LIN {X 0,Y 573.248,Z 41.082,A -85,B 0,C 180,E1 -2299.475,E2 -2299.475} C_VEL
LIN {X 0,Y 573.238,Z 41.075,A -85,B 0,C 180,E1 -2302.192,E2 -2302.192} C_VEL
LIN {X 0,Y 573.24,Z 41.084,A -85,B 0,C 180,E1 -2305.229,E2 -2305.229} C_VEL
LIN {X 0,Y 573.243,Z 41.074,A -85,B 0,C 180,E1 -2308.185,E2 -2308.185} C_VEL
LIN {X 0,Y 573.268,Z 41.074,A -85,B 0,C 180,E1 -2310.634,E2 -2310.634} C_VEL
LIN {X 0,Y 573.255,Z 41.08,A -85,B 0,C 180,E1 -2313.024,E2 -2313.024} C_VEL
LIN {X 0,Y 573.279,Z 41.072,A -85,B 0,C 180,E1 -2315.366,E2 -2315.366} C_VEL
LIN {X 0,Y 573.234,Z 41.08,A -85,B 0,C 180,E1 -2318.419,E2 -2318.419} C_VEL
LIN {X 0,Y 573.274,Z 41.078,A -85,B 0,C 180,E1 -2320.731,E2 -2320.731} C_VEL
LIN {X 0,Y 573.252,Z 41.072,A -85,B 0,C 180,E1 -2323.622,E2 -2323.622} C_VEL
LIN {X 0,Y 573.277,Z 41.072,A -85,B 0,C 180,E1 -2325.807,E2 -2325.807} C_VEL
LIN {X 0,Y 573.269,Z 41.074,A -85,B 0,C 180,E1 -2328.745,E2 -2328.745} C_VEL
LIN {X 0,Y 573.288,Z 41.07,A -85,B 0,C 180,E1 -2331.54,E2 -2331.54} C_VEL
LIN {X 0,Y 573.29,Z 41.073,A -85,B 0,C 180,E1 -2334.372,E2 -2334.372} C_VEL
LIN {X 0,Y 573.311,Z 41.074,A -85,B 0,C 180,E1 -2337.892,E2 -2337.892} C_VEL
LIN {X 0,Y 573.332,Z 41.063,A -85,B 0,C 180,E1 -2340.702,E2 -2340.702} C_VEL
LIN {X 0,Y 573.234,Z 41.082,A -85,B 0,C 180,E1 -2343.514,E2 -2343.514} C_VEL
LIN {X 0,Y 573.286,Z 41.078,A -85,B 0,C 180,E1 -2345.628,E2 -2345.628} C_VEL
LIN {X 0,Y 573.275,Z 41.075,A -85,B 0,C 180,E1 -2347.75,E2 -2347.75} C_VEL
LIN {X 0,Y 573.267,Z 41.071,A -85,B 0,C 180,E1 -2350.597,E2 -2350.597} C_VEL
LIN {X 0,Y 573.266,Z 41.073,A -85,B 0,C 180,E1 -2352.748,E2 -2352.748} C_VEL
LIN {X 0,Y 573.239,Z 41.079,A -85,B 0,C 180,E1 -2354.92,E2 -2354.92} C_VEL
LIN {X 0,Y 573.242,Z 41.074,A -85,B 0,C 180,E1 -2357.849,E2 -2357.849} C_VEL
LIN {X 0,Y 573.244,Z 41.074,A -85,B 0,C 180,E1 -2360.077,E2 -2360.077} C_VEL
LIN {X 0,Y 573.236,Z 41.077,A -85,B 0,C 180,E1 -2362.338,E2 -2362.338} C_VEL
LIN {X 0,Y 573.249,Z 41.076,A -85,B 0,C 180,E1 -2364.376,E2 -2364.376} C_VEL
LIN {X 0,Y 572.619,Z 41.161,A -85,B 0,C 180,E1 -2364.962,E2 -2364.962} C_VEL
LIN {X 0,Y 569.76,Z 41.516,A -85,B 0,C 180,E1 -2365.913,E2 -2365.913} C_VEL
LIN {X 0,Y 567.316,Z 41.821,A -85,B 0,C 180,E1 -2366.679,E2 -2366.679} C_VEL
LIN {X 0,Y 566.259,Z 41.946,A -85,B 0,C 180,E1 -2367.27,E2 -2367.27} C_VEL
LIN {X 0,Y 566.171,Z 41.955,A -85,B 0,C 180,E1 -2367.47,E2 -2367.47} C_VEL
LIN {X 0,Y 566.203,Z 41.952,A -85,B 0,C 180,E1 -2369.769,E2 -2369.769} C_VEL
LIN {X 0,Y 566.206,Z 41.959,A -85,B 0,C 180,E1 -2372.43,E2 -2372.43} C_VEL
LIN {X 0,Y 566.172,Z 41.957,A -85,B 0,C 180,E1 -2374.988,E2 -2374.988} C_VEL
LIN {X 0,Y 566.194,Z 41.952,A -85,B 0,C 180,E1 -2377.461,E2 -2377.461} C_VEL
LIN {X 0,Y 566.209,Z 41.957,A -85,B 0,C 180,E1 -2380.199,E2 -2380.199} C_VEL
LIN {X 0,Y 566.197,Z 41.953,A -85,B 0,C 180,E1 -2383.055,E2 -2383.055} C_VEL
LIN {X 0,Y 566.161,Z 41.965,A -85,B 0,C 180,E1 -2386.053,E2 -2386.053} C_VEL
LIN {X 0,Y 566.172,Z 41.956,A -85,B 0,C 180,E1 -2388.86,E2 -2388.86} C_VEL
LIN {X 0,Y 566.204,Z 41.957,A -85,B 0,C 180,E1 -2391.443,E2 -2391.443} C_VEL
LIN {X 0,Y 566.151,Z 41.96,A -85,B 0,C 180,E1 -2394.307,E2 -2394.307} C_VEL
LIN {X 0,Y 566.2,Z 41.955,A -85,B 0,C 180,E1 -2396.896,E2 -2396.896} C_VEL
LIN {X 0,Y 566.17,Z 41.965,A -85,B 0,C 180,E1 -2399.406,E2 -2399.406} C_VEL
LIN {X 0,Y 566.248,Z 42.03,A -85,B 0,C 180,E1 -2402.287,E2 -2402.287} C_VEL
LIN {X 0,Y 566.323,Z 51.031,A -85,B 0,C 180,E1 -2404.059,E2 -2404.059} C_VEL
LIN {X 0,Y 566.238,Z 61.144,A -85,B 0,C 180,E1 -2406.046,E2 -2406.046} C_VEL
LIN {X 0,Y 567.205,Z 67.037,A -85,B 0,C 180,E1 -2406.16,E2 -2406.16} C_VEL
LIN {X 0,Y 566.926,Z 167.119,A -85,B 0,C 180,E1 -2407.448,E2 -2407.448} C_VEL
LIN {X 0,Y 566.828,Z 180.881,A -85,B 0,C 180,E1 -2407.78,E2 -2407.78} C_VEL
LIN {X 0,Y 566.748,Z 192.877,A -85,B 0,C 180,E1 -2408.21,E2 -2408.21} C_VEL
LIN {X 0,Y 566.57,Z 204.986,A -85,B 0,C 180,E1 -2408.797,E2 -2408.797} C_VEL
LIN {X 0,Y 566.416,Z 215.924,A -85,B 0,C 180,E1 -2409.481,E2 -2409.481} C_VEL
LIN {X 0,Y 566.302,Z 226.819,A -85,B 0,C 180,E1 -2410.328,E2 -2410.328} C_VEL
LIN {X 0,Y 566.23,Z 235.633,A -85,B 0,C 180,E1 -2411.173,E2 -2411.173} C_VEL
LIN {X 0,Y 566.102,Z 243.65,A -85,B 0,C 180,E1 -2412.105,E2 -2412.105} C_VEL
LIN {X 0,Y 566.039,Z 251.146,A -85,B 0,C 180,E1 -2413.176,E2 -2413.176} C_VEL
LIN {X 0,Y 565.951,Z 256.676,A -85,B 0,C 180,E1 -2414.145,E2 -2414.145} C_VEL
LIN {X 0,Y 565.943,Z 261.72,A -85,B 0,C 180,E1 -2415.252,E2 -2415.252} C_VEL
LIN {X 0,Y 565.899,Z 265.562,A -85,B 0,C 180,E1 -2416.351,E2 -2416.351} C_VEL
LIN {X 0,Y 565.86,Z 267.528,A -85,B 0,C 180,E1 -2417.082,E2 -2417.082} C_VEL
LIN {X 0,Y 565.869,Z 269.041,A -85,B 0,C 180,E1 -2417.811,E2 -2417.811} C_VEL
LIN {X 0,Y 565.901,Z 270.434,A -85,B 0,C 180,E1 -2418.846,E2 -2418.846} C_VEL
LIN {X 0,Y 565.882,Z 270.993,A -85,B 0,C 180,E1 -2419.987,E2 -2419.987} C_VEL
LIN {X 0,Y 565.829,Z 270.818,A -85,B 0,C 180,E1 -2420.708,E2 -2420.708} C_VEL
LIN {X 0,Y 565.851,Z 270.228,A -85,B 0,C 180,E1 -2421.429,E2 -2421.429} C_VEL
LIN {X 0,Y 565.877,Z 269.245,A -85,B 0,C 180,E1 -2422.148,E2 -2422.148} C_VEL
LIN {X 0,Y 565.945,Z 266.439,A -85,B 0,C 180,E1 -2423.44,E2 -2423.44} C_VEL
LIN {X 0,Y 565.921,Z 262.45,A -85,B 0,C 180,E1 -2424.656,E2 -2424.656} C_VEL
LIN {X 0,Y 565.964,Z 257.776,A -85,B 0,C 180,E1 -2425.727,E2 -2425.727} C_VEL
LIN {X 0,Y 566.004,Z 250.768,A -85,B 0,C 180,E1 -2426.975,E2 -2426.975} C_VEL
LIN {X 0,Y 566.065,Z 243.204,A -85,B 0,C 180,E1 -2428.043,E2 -2428.043} C_VEL
LIN {X 0,Y 566.211,Z 233.725,A -85,B 0,C 180,E1 -2429.111,E2 -2429.111} C_VEL
LIN {X 0,Y 566.297,Z 223.997,A -85,B 0,C 180,E1 -2430,E2 -2430} C_VEL
LIN {X 0,Y 566.443,Z 213.138,A -85,B 0,C 180,E1 -2430.8,E2 -2430.8} C_VEL
LIN {X 0,Y 566.657,Z 200.84,A -85,B 0,C 180,E1 -2431.51,E2 -2431.51} C_VEL
LIN {X 0,Y 566.769,Z 188.815,A -85,B 0,C 180,E1 -2432.043,E2 -2432.043} C_VEL
LIN {X 0,Y 566.841,Z 176.197,A -85,B 0,C 180,E1 -2432.443,E2 -2432.443} C_VEL
LIN {X 0,Y 566.958,Z 162.831,A -85,B 0,C 180,E1 -2432.709,E2 -2432.709} C_VEL
LIN {X 0,Y 567.076,Z 66.314,A -85,B 0,C 180,E1 -2433.942,E2 -2433.942} C_VEL
LIN {X 0,Y 566.213,Z 61.132,A -85,B 0,C 180,E1 -2434.048,E2 -2434.048} C_VEL
LIN {X 0,Y 566.361,Z 48.01,A -85,B 0,C 180,E1 -2436.625,E2 -2436.625} C_VEL
LIN {X 0,Y 566.229,Z 41.953,A -85,B 0,C 180,E1 -2437.847,E2 -2437.847} C_VEL
LIN {X 0,Y 566.24,Z 41.956,A -85,B 0,C 180,E1 -2440.73,E2 -2440.73} C_VEL
LIN {X 0,Y 566.21,Z 41.955,A -85,B 0,C 180,E1 -2442.91,E2 -2442.91} C_VEL
LIN {X 0,Y 566.201,Z 41.953,A -85,B 0,C 180,E1 -2445.11,E2 -2445.11} C_VEL
LIN {X 0,Y 566.202,Z 41.951,A -85,B 0,C 180,E1 -2447.332,E2 -2447.332} C_VEL
LIN {X 0,Y 566.21,Z 41.96,A -85,B 0,C 180,E1 -2450.338,E2 -2450.338} C_VEL
LIN {X 0,Y 566.171,Z 41.955,A -85,B 0,C 180,E1 -2453.281,E2 -2453.281} C_VEL
LIN {X 0,Y 566.215,Z 41.953,A -85,B 0,C 180,E1 -2455.749,E2 -2455.749} C_VEL
LIN {X 0,Y 566.205,Z 41.958,A -85,B 0,C 180,E1 -2458.202,E2 -2458.202} C_VEL
LIN {X 0,Y 566.193,Z 41.952,A -85,B 0,C 180,E1 -2461.077,E2 -2461.077} C_VEL
LIN {X 0,Y 566.215,Z 41.957,A -85,B 0,C 180,E1 -2463.734,E2 -2463.734} C_VEL
LIN {X 0,Y 566.21,Z 41.951,A -85,B 0,C 180,E1 -2466.57,E2 -2466.57} C_VEL
LIN {X 0,Y 566.219,Z 41.959,A -85,B 0,C 180,E1 -2469.686,E2 -2469.686} C_VEL
LIN {X 0,Y 566.204,Z 41.952,A -85,B 0,C 180,E1 -2472.917,E2 -2472.917} C_VEL
LIN {X 0,Y 566.197,Z 41.953,A -85,B 0,C 180,E1 -2476.05,E2 -2476.05} C_VEL
LIN {X 0,Y 566.207,Z 41.958,A -85,B 0,C 180,E1 -2479.215,E2 -2479.215} C_VEL
LIN {X 0,Y 566.189,Z 41.956,A -85,B 0,C 180,E1 -2481.637,E2 -2481.637} C_VEL
LIN {X 0,Y 566.167,Z 41.956,A -85,B 0,C 180,E1 -2484.308,E2 -2484.308} C_VEL
LIN {X 0,Y 566.224,Z 41.956,A -85,B 0,C 180,E1 -2486.898,E2 -2486.898} C_VEL
LIN {X 0,Y 566.185,Z 41.956,A -85,B 0,C 180,E1 -2489.407,E2 -2489.407} C_VEL
LIN {X 0,Y 566.217,Z 41.949,A -85,B 0,C 180,E1 -2491.858,E2 -2491.858} C_VEL
LIN {X 0,Y 566.214,Z 41.952,A -85,B 0,C 180,E1 -2494.251,E2 -2494.251} C_VEL
LIN {X 0,Y 566.178,Z 41.964,A -85,B 0,C 180,E1 -2496.719,E2 -2496.719} C_VEL
LIN {X 0,Y 566.212,Z 41.95,A -85,B 0,C 180,E1 -2499.663,E2 -2499.663} C_VEL
LIN {X 0,Y 566.203,Z 41.957,A -85,B 0,C 180,E1 -2502.669,E2 -2502.669} C_VEL
LIN {X 0,Y 566.24,Z 41.947,A -85,B 0,C 180,E1 -2505.627,E2 -2505.627} C_VEL
LIN {X 0,Y 566.241,Z 41.95,A -85,B 0,C 180,E1 -2508.675,E2 -2508.675} C_VEL
LIN {X 0,Y 566.212,Z 41.951,A -85,B 0,C 180,E1 -2511.434,E2 -2511.434} C_VEL
LIN {X 0,Y 566.259,Z 41.95,A -85,B 0,C 180,E1 -2514.302,E2 -2514.302} C_VEL
LIN {X 0,Y 566.284,Z 41.95,A -85,B 0,C 180,E1 -2517.866,E2 -2517.866} C_VEL
LIN {X 0,Y 566.304,Z 41.939,A -85,B 0,C 180,E1 -2520.711,E2 -2520.711} C_VEL
LIN {X 0,Y 566.273,Z 41.942,A -85,B 0,C 180,E1 -2522.846,E2 -2522.846} C_VEL
LIN {X 0,Y 566.255,Z 41.953,A -85,B 0,C 180,E1 -2525.698,E2 -2525.698} C_VEL
LIN {X 0,Y 566.211,Z 41.95,A -85,B 0,C 180,E1 -2528.566,E2 -2528.566} C_VEL
LIN {X 0,Y 566.248,Z 41.955,A -85,B 0,C 180,E1 -2531.454,E2 -2531.454} C_VEL
LIN {X 0,Y 566.236,Z 41.947,A -85,B 0,C 180,E1 -2534.504,E2 -2534.504} C_VEL
LIN {X 0,Y 566.204,Z 41.959,A -85,B 0,C 180,E1 -2537.332,E2 -2537.332} C_VEL
LIN {X 0,Y 566.212,Z 41.95,A -85,B 0,C 180,E1 -2540.337,E2 -2540.337} C_VEL
LIN {X 0,Y 566.174,Z 41.96,A -85,B 0,C 180,E1 -2543.281,E2 -2543.281} C_VEL
LIN {X 0,Y 566.211,Z 41.95,A -85,B 0,C 180,E1 -2545.749,E2 -2545.749} C_VEL
LIN {X 0,Y 566.209,Z 41.952,A -85,B 0,C 180,E1 -2548.202,E2 -2548.202} C_VEL
LIN {X 0,Y 566.195,Z 41.956,A -85,B 0,C 180,E1 -2551.076,E2 -2551.076} C_VEL
LIN {X 0,Y 566.201,Z 41.951,A -85,B 0,C 180,E1 -2553.732,E2 -2553.732} C_VEL
LIN {X 0,Y 566.187,Z 41.962,A -85,B 0,C 180,E1 -2556.571,E2 -2556.571} C_VEL
LIN {X 0,Y 566.218,Z 41.95,A -85,B 0,C 180,E1 -2559.685,E2 -2559.685} C_VEL
LIN {X 0,Y 566.205,Z 41.952,A -85,B 0,C 180,E1 -2562.917,E2 -2562.917} C_VEL
LIN {X 0,Y 566.164,Z 41.962,A -85,B 0,C 180,E1 -2565.96,E2 -2565.96} C_VEL
LIN {X 0,Y 566.19,Z 41.962,A -85,B 0,C 180,E1 -2568.139,E2 -2568.139} C_VEL
LIN {X 0,Y 566.214,Z 41.95,A -85,B 0,C 180,E1 -2570.726,E2 -2570.726} C_VEL
LIN {X 0,Y 566.186,Z 41.956,A -85,B 0,C 180,E1 -2573.429,E2 -2573.429} C_VEL
LIN {X 0,Y 566.201,Z 41.954,A -85,B 0,C 180,E1 -2576.268,E2 -2576.268} C_VEL
LIN {X 0,Y 566.191,Z 41.953,A -85,B 0,C 180,E1 -2578.924,E2 -2578.924} C_VEL
LIN {X 0,Y 566.216,Z 41.956,A -85,B 0,C 180,E1 -2581.857,E2 -2581.857} C_VEL
LIN {X 0,Y 566.21,Z 41.953,A -85,B 0,C 180,E1 -2584.251,E2 -2584.251} C_VEL
LIN {X 0,Y 566.261,Z 42.121,A -85,B 0,C 180,E1 -2585.676,E2 -2585.676} C_VEL
LIN {X 0,Y 567.074,Z 47.877,A -85,B 0,C 180,E1 -2586.508,E2 -2586.508} C_VEL
LIN {X 0,Y 566.844,Z 66.903,A -85,B 0,C 180,E1 -2589.117,E2 -2589.117} C_VEL
LIN {X 0,Y 566.689,Z 87.816,A -85,B 0,C 180,E1 -2591.938,E2 -2591.938} C_VEL
LIN {X 0,Y 566.434,Z 110.041,A -85,B 0,C 180,E1 -2594.897,E2 -2594.897} C_VEL
LIN {X 0,Y 566.431,Z 118.274,A -85,B 0,C 180,E1 -2595.987,E2 -2595.987} C_VEL
LIN {X 0,Y 567.176,Z 125.162,A -85,B 0,C 180,E1 -2596.095,E2 -2596.095} C_VEL
LIN {X 0,Y 566.941,Z 226.937,A -85,B 0,C 180,E1 -2597.402,E2 -2597.402} C_VEL
LIN {X 0,Y 566.859,Z 240.211,A -85,B 0,C 180,E1 -2597.719,E2 -2597.719} C_VEL
LIN {X 0,Y 566.761,Z 252.373,A -85,B 0,C 180,E1 -2598.148,E2 -2598.148} C_VEL
LIN {X 0,Y 566.604,Z 264.236,A -85,B 0,C 180,E1 -2598.712,E2 -2598.712} C_VEL
LIN {X 0,Y 566.442,Z 276.192,A -85,B 0,C 180,E1 -2599.455,E2 -2599.455} C_VEL
LIN {X 0,Y 566.325,Z 286.604,A -85,B 0,C 180,E1 -2600.265,E2 -2600.265} C_VEL
LIN {X 0,Y 566.207,Z 295.112,A -85,B 0,C 180,E1 -2601.074,E2 -2601.074} C_VEL
LIN {X 0,Y 566.112,Z 302.96,A -85,B 0,C 180,E1 -2601.972,E2 -2601.972} C_VEL
LIN {X 0,Y 566.004,Z 310.622,A -85,B 0,C 180,E1 -2603.047,E2 -2603.047} C_VEL
LIN {X 0,Y 566.004,Z 317.679,A -85,B 0,C 180,E1 -2604.299,E2 -2604.299} C_VEL
LIN {X 0,Y 565.933,Z 322.372,A -85,B 0,C 180,E1 -2605.37,E2 -2605.37} C_VEL
LIN {X 0,Y 565.927,Z 325.958,A -85,B 0,C 180,E1 -2606.44,E2 -2606.44} C_VEL
LIN {X 0,Y 565.878,Z 327.807,A -85,B 0,C 180,E1 -2607.152,E2 -2607.152} C_VEL
LIN {X 0,Y 565.846,Z 330.183,A -85,B 0,C 180,E1 -2608.577,E2 -2608.577} C_VEL
LIN {X 0,Y 565.839,Z 331,A -85,B 0,C 180,E1 -2610,E2 -2610} C_VEL
LIN {X 0,Y 565.846,Z 330.185,A -85,B 0,C 180,E1 -2611.423,E2 -2611.423} C_VEL
LIN {X 0,Y 565.878,Z 327.81,A -85,B 0,C 180,E1 -2612.848,E2 -2612.848} C_VEL
LIN {X 0,Y 565.926,Z 324.895,A -85,B 0,C 180,E1 -2613.916,E2 -2613.916} C_VEL
LIN {X 0,Y 565.878,Z 320.948,A -85,B 0,C 180,E1 -2614.987,E2 -2614.987} C_VEL
LIN {X 0,Y 566.004,Z 315.867,A -85,B 0,C 180,E1 -2616.058,E2 -2616.058} C_VEL
LIN {X 0,Y 566.04,Z 309.467,A -85,B 0,C 180,E1 -2617.132,E2 -2617.132} C_VEL
LIN {X 0,Y 566.134,Z 301.477,A -85,B 0,C 180,E1 -2618.208,E2 -2618.208} C_VEL
LIN {X 0,Y 566.229,Z 293.333,A -85,B 0,C 180,E1 -2619.105,E2 -2619.105} C_VEL
LIN {X 0,Y 566.342,Z 283.397,A -85,B 0,C 180,E1 -2620.005,E2 -2620.005} C_VEL
LIN {X 0,Y 566.512,Z 272.289,A -85,B 0,C 180,E1 -2620.808,E2 -2620.808} C_VEL
LIN {X 0,Y 566.613,Z 261.17,A -85,B 0,C 180,E1 -2621.447,E2 -2621.447} C_VEL
LIN {X 0,Y 566.748,Z 248.975,A -85,B 0,C 180,E1 -2621.988,E2 -2621.988} C_VEL
LIN {X 0,Y 566.887,Z 236.171,A -85,B 0,C 180,E1 -2622.394,E2 -2622.394} C_VEL
LIN {X 0,Y 566.991,Z 224.1,A -85,B 0,C 180,E1 -2622.642,E2 -2622.642} C_VEL
LIN {X 0,Y 567.07,Z 122.848,A -85,B 0,C 180,E1 -2623.937,E2 -2623.937} C_VEL
LIN {X 0,Y 566.43,Z 118.181,A -85,B 0,C 180,E1 -2624.024,E2 -2624.024} C_VEL
LIN {X 0,Y 566.583,Z 96.455,A -85,B 0,C 180,E1 -2626.903,E2 -2626.903} C_VEL
LIN {X 0,Y 566.791,Z 75.206,A -85,B 0,C 180,E1 -2629.748,E2 -2629.748} C_VEL
LIN {X 0,Y 566.965,Z 54.285,A -85,B 0,C 180,E1 -2632.599,E2 -2632.599} C_VEL
LIN {X 0,Y 566.958,Z 45.846,A -85,B 0,C 180,E1 -2633.766,E2 -2633.766} C_VEL
LIN {X 0,Y 566.257,Z 41.954,A -85,B 0,C 180,E1 -2634.349,E2 -2634.349} C_VEL
LIN {X 0,Y 566.211,Z 41.952,A -85,B 0,C 180,E1 -2637.339,E2 -2637.339} C_VEL
LIN {X 0,Y 566.204,Z 41.954,A -85,B 0,C 180,E1 -2639.769,E2 -2639.769} C_VEL
LIN {X 0,Y 566.206,Z 41.957,A -85,B 0,C 180,E1 -2642.43,E2 -2642.43} C_VEL
LIN {X 0,Y 566.184,Z 41.954,A -85,B 0,C 180,E1 -2644.99,E2 -2644.99} C_VEL
LIN {X 0,Y 566.199,Z 41.954,A -85,B 0,C 180,E1 -2647.461,E2 -2647.461} C_VEL
LIN {X 0,Y 566.21,Z 41.955,A -85,B 0,C 180,E1 -2650.199,E2 -2650.199} C_VEL
LIN {X 0,Y 566.203,Z 41.952,A -85,B 0,C 180,E1 -2653.054,E2 -2653.054} C_VEL
LIN {X 0,Y 566.197,Z 41.955,A -85,B 0,C 180,E1 -2656.049,E2 -2656.049} C_VEL
LIN {X 0,Y 566.207,Z 41.955,A -85,B 0,C 180,E1 -2659.215,E2 -2659.215} C_VEL
LIN {X 0,Y 566.189,Z 41.958,A -85,B 0,C 180,E1 -2661.637,E2 -2661.637} C_VEL
LIN {X 0,Y 566.167,Z 41.955,A -85,B 0,C 180,E1 -2664.308,E2 -2664.308} C_VEL
LIN {X 0,Y 566.207,Z 41.955,A -85,B 0,C 180,E1 -2666.897,E2 -2666.897} C_VEL
LIN {X 0,Y 566.185,Z 41.957,A -85,B 0,C 180,E1 -2669.407,E2 -2669.407} C_VEL
LIN {X 0,Y 566.217,Z 41.95,A -85,B 0,C 180,E1 -2671.857,E2 -2671.857} C_VEL
LIN {X 0,Y 566.214,Z 41.95,A -85,B 0,C 180,E1 -2674.251,E2 -2674.251} C_VEL
LIN {X 0,Y 566.174,Z 41.964,A -85,B 0,C 180,E1 -2676.719,E2 -2676.719} C_VEL
LIN {X 0,Y 566.212,Z 41.95,A -85,B 0,C 180,E1 -2679.663,E2 -2679.663} C_VEL
LIN {X 0,Y 566.203,Z 41.957,A -85,B 0,C 180,E1 -2682.668,E2 -2682.668} C_VEL
LIN {X 0,Y 566.239,Z 41.947,A -85,B 0,C 180,E1 -2685.627,E2 -2685.627} C_VEL
LIN {X 0,Y 566.241,Z 41.95,A -85,B 0,C 180,E1 -2688.675,E2 -2688.675} C_VEL
LIN {X 0,Y 566.232,Z 41.948,A -85,B 0,C 180,E1 -2691.434,E2 -2691.434} C_VEL
LIN {X 0,Y 566.259,Z 41.95,A -85,B 0,C 180,E1 -2694.302,E2 -2694.302} C_VEL
LIN {X 0,Y 566.283,Z 41.949,A -85,B 0,C 180,E1 -2697.866,E2 -2697.866} C_VEL
LIN {X 0,Y 566.303,Z 41.939,A -85,B 0,C 180,E1 -2700.711,E2 -2700.711} C_VEL
LIN {X 0,Y 566.272,Z 41.942,A -85,B 0,C 180,E1 -2702.845,E2 -2702.845} C_VEL
LIN {X 0,Y 566.253,Z 41.953,A -85,B 0,C 180,E1 -2705.698,E2 -2705.698} C_VEL
LIN {X 0,Y 566.209,Z 41.949,A -85,B 0,C 180,E1 -2708.566,E2 -2708.566} C_VEL
LIN {X 0,Y 566.247,Z 41.954,A -85,B 0,C 180,E1 -2711.454,E2 -2711.454} C_VEL
LIN {X 0,Y 566.234,Z 41.947,A -85,B 0,C 180,E1 -2714.504,E2 -2714.504} C_VEL
LIN {X 0,Y 566.202,Z 41.957,A -85,B 0,C 180,E1 -2717.332,E2 -2717.332} C_VEL
LIN {X 0,Y 566.211,Z 41.951,A -85,B 0,C 180,E1 -2720.337,E2 -2720.337} C_VEL
LIN {X 0,Y 566.172,Z 41.958,A -85,B 0,C 180,E1 -2723.28,E2 -2723.28} C_VEL
LIN {X 0,Y 566.208,Z 41.951,A -85,B 0,C 180,E1 -2725.749,E2 -2725.749} C_VEL
LIN {X 0,Y 566.171,Z 41.955,A -85,B 0,C 180,E1 -2727.47,E2 -2727.47} C_VEL
LIN {X 0,Y 565.5,Z 42.041,A -85,B 0,C 180,E1 -2728.064,E2 -2728.064} C_VEL
LIN {X 0,Y 562.649,Z 42.398,A -85,B 0,C 180,E1 -2729.028,E2 -2729.028} C_VEL
LIN {X 0,Y 560.247,Z 42.696,A -85,B 0,C 180,E1 -2729.804,E2 -2729.804} C_VEL
LIN {X 0,Y 559.221,Z 42.828,A -85,B 0,C 180,E1 -2730.403,E2 -2730.403} C_VEL
LIN {X 0,Y 559.141,Z 42.832,A -85,B 0,C 180,E1 -2730.606,E2 -2730.606} C_VEL
LIN {X 0,Y 559.156,Z 42.835,A -85,B 0,C 180,E1 -2732.715,E2 -2732.715} C_VEL
LIN {X 0,Y 559.121,Z 42.834,A -85,B 0,C 180,E1 -2735.325,E2 -2735.325} C_VEL
LIN {X 0,Y 559.132,Z 42.837,A -85,B 0,C 180,E1 -2738.018,E2 -2738.018} C_VEL
LIN {X 0,Y 559.156,Z 42.828,A -85,B 0,C 180,E1 -2740.812,E2 -2740.812} C_VEL
LIN {X 0,Y 559.138,Z 42.837,A -85,B 0,C 180,E1 -2743.734,E2 -2743.734} C_VEL
LIN {X 0,Y 559.133,Z 42.833,A -85,B 0,C 180,E1 -2746.805,E2 -2746.805} C_VEL
LIN {X 0,Y 559.157,Z 42.831,A -85,B 0,C 180,E1 -2749.187,E2 -2749.187} C_VEL
LIN {X 0,Y 559.127,Z 42.839,A -85,B 0,C 180,E1 -2751.982,E2 -2751.982} C_VEL
LIN {X 0,Y 559.13,Z 42.834,A -85,B 0,C 180,E1 -2754.788,E2 -2754.788} C_VEL
LIN {X 0,Y 559.154,Z 42.839,A -85,B 0,C 180,E1 -2757.365,E2 -2757.365} C_VEL
LIN {X 0,Y 559.12,Z 42.837,A -85,B 0,C 180,E1 -2760.148,E2 -2760.148} C_VEL
LIN {X 0,Y 559.225,Z 42.921,A -85,B 0,C 180,E1 -2762.19,E2 -2762.19} C_VEL
LIN {X 0,Y 559.332,Z 49.619,A -85,B 0,C 180,E1 -2763.524,E2 -2763.524} C_VEL
LIN {X 0,Y 559.216,Z 61.527,A -85,B 0,C 180,E1 -2765.878,E2 -2765.878} C_VEL
LIN {X 0,Y 560.309,Z 68.487,A -85,B 0,C 180,E1 -2766,E2 -2766} C_VEL
LIN {X 0,Y 559.997,Z 167.977,A -85,B 0,C 180,E1 -2767.299,E2 -2767.299} C_VEL
LIN {X 0,Y 559.923,Z 181.603,A -85,B 0,C 180,E1 -2767.637,E2 -2767.637} C_VEL
LIN {X 0,Y 559.809,Z 193.573,A -85,B 0,C 180,E1 -2768.075,E2 -2768.075} C_VEL
LIN {X 0,Y 559.626,Z 205.125,A -85,B 0,C 180,E1 -2768.642,E2 -2768.642} C_VEL
LIN {X 0,Y 559.456,Z 215.753,A -85,B 0,C 180,E1 -2769.31,E2 -2769.31} C_VEL
LIN {X 0,Y 559.327,Z 226.671,A -85,B 0,C 180,E1 -2770.168,E2 -2770.168} C_VEL
LIN {X 0,Y 559.208,Z 236.374,A -85,B 0,C 180,E1 -2771.118,E2 -2771.118} C_VEL
LIN {X 0,Y 559.039,Z 244.23,A -85,B 0,C 180,E1 -2772.061,E2 -2772.061} C_VEL
LIN {X 0,Y 558.957,Z 251.861,A -85,B 0,C 180,E1 -2773.191,E2 -2773.191} C_VEL
LIN {X 0,Y 558.865,Z 257.92,A -85,B 0,C 180,E1 -2774.313,E2 -2774.313} C_VEL
LIN {X 0,Y 558.826,Z 263.113,A -85,B 0,C 180,E1 -2775.554,E2 -2775.554} C_VEL
LIN {X 0,Y 558.763,Z 267.208,A -85,B 0,C 180,E1 -2776.915,E2 -2776.915} C_VEL
LIN {X 0,Y 558.777,Z 268.806,A -85,B 0,C 180,E1 -2777.654,E2 -2777.654} C_VEL
LIN {X 0,Y 558.798,Z 270.417,A -85,B 0,C 180,E1 -2778.815,E2 -2778.815} C_VEL
LIN {X 0,Y 558.778,Z 270.965,A -85,B 0,C 180,E1 -2779.858,E2 -2779.858} C_VEL
LIN {X 0,Y 558.74,Z 270.885,A -85,B 0,C 180,E1 -2780.589,E2 -2780.589} C_VEL
LIN {X 0,Y 558.765,Z 270.368,A -85,B 0,C 180,E1 -2781.319,E2 -2781.319} C_VEL
LIN {X 0,Y 558.795,Z 269.441,A -85,B 0,C 180,E1 -2782.048,E2 -2782.048} C_VEL
LIN {X 0,Y 558.844,Z 266.487,A -85,B 0,C 180,E1 -2783.464,E2 -2783.464} C_VEL
LIN {X 0,Y 558.845,Z 262.934,A -85,B 0,C 180,E1 -2784.588,E2 -2784.588} C_VEL
LIN {X 0,Y 558.892,Z 258.419,A -85,B 0,C 180,E1 -2785.673,E2 -2785.673} C_VEL
LIN {X 0,Y 558.911,Z 251.637,A -85,B 0,C 180,E1 -2786.937,E2 -2786.937} C_VEL
LIN {X 0,Y 559,Z 244.308,A -85,B 0,C 180,E1 -2788.019,E2 -2788.019} C_VEL
LIN {X 0,Y 559.167,Z 236.838,A -85,B 0,C 180,E1 -2788.92,E2 -2788.92} C_VEL
LIN {X 0,Y 559.265,Z 227.84,A -85,B 0,C 180,E1 -2789.82,E2 -2789.82} C_VEL
LIN {X 0,Y 559.394,Z 217.864,A -85,B 0,C 180,E1 -2790.63,E2 -2790.63} C_VEL
LIN {X 0,Y 559.62,Z 206.803,A -85,B 0,C 180,E1 -2791.349,E2 -2791.349} C_VEL
LIN {X 0,Y 559.803,Z 194.425,A -85,B 0,C 180,E1 -2791.979,E2 -2791.979} C_VEL
LIN {X 0,Y 559.895,Z 181.704,A -85,B 0,C 180,E1 -2792.451,E2 -2792.451} C_VEL
LIN {X 0,Y 560.034,Z 168.079,A -85,B 0,C 180,E1 -2792.787,E2 -2792.787} C_VEL
LIN {X 0,Y 560.184,Z 66.835,A -85,B 0,C 180,E1 -2794.114,E2 -2794.114} C_VEL
LIN {X 0,Y 559.194,Z 61.429,A -85,B 0,C 180,E1 -2794.235,E2 -2794.235} C_VEL
LIN {X 0,Y 559.377,Z 48.905,A -85,B 0,C 180,E1 -2796.705,E2 -2796.705} C_VEL
LIN {X 0,Y 559.206,Z 42.829,A -85,B 0,C 180,E1 -2797.924,E2 -2797.924} C_VEL
LIN {X 0,Y 559.197,Z 42.831,A -85,B 0,C 180,E1 -2800.867,E2 -2800.867} C_VEL
LIN {X 0,Y 559.173,Z 42.827,A -85,B 0,C 180,E1 -2803.816,E2 -2803.816} C_VEL
LIN {X 0,Y 559.183,Z 42.83,A -85,B 0,C 180,E1 -2806.803,E2 -2806.803} C_VEL
LIN {X 0,Y 559.168,Z 42.829,A -85,B 0,C 180,E1 -2809.838,E2 -2809.838} C_VEL
LIN {X 0,Y 559.144,Z 42.838,A -85,B 0,C 180,E1 -2812.153,E2 -2812.153} C_VEL
LIN {X 0,Y 559.178,Z 42.826,A -85,B 0,C 180,E1 -2815.298,E2 -2815.298} C_VEL
LIN {X 0,Y 559.184,Z 42.829,A -85,B 0,C 180,E1 -2817.712,E2 -2817.712} C_VEL
LIN {X 0,Y 559.156,Z 42.836,A -85,B 0,C 180,E1 -2820.183,E2 -2820.183} C_VEL
LIN {X 0,Y 559.159,Z 42.829,A -85,B 0,C 180,E1 -2822.715,E2 -2822.715} C_VEL
LIN {X 0,Y 559.147,Z 42.832,A -85,B 0,C 180,E1 -2825.323,E2 -2825.323} C_VEL
LIN {X 0,Y 559.135,Z 42.836,A -85,B 0,C 180,E1 -2828.018,E2 -2828.018} C_VEL
LIN {X 0,Y 559.158,Z 42.829,A -85,B 0,C 180,E1 -2830.813,E2 -2830.813} C_VEL
LIN {X 0,Y 559.141,Z 42.837,A -85,B 0,C 180,E1 -2833.734,E2 -2833.734} C_VEL
LIN {X 0,Y 559.148,Z 42.831,A -85,B 0,C 180,E1 -2836.804,E2 -2836.804} C_VEL
LIN {X 0,Y 559.159,Z 42.836,A -85,B 0,C 180,E1 -2839.188,E2 -2839.188} C_VEL
LIN {X 0,Y 559.136,Z 42.832,A -85,B 0,C 180,E1 -2841.983,E2 -2841.983} C_VEL
LIN {X 0,Y 559.137,Z 42.836,A -85,B 0,C 180,E1 -2844.787,E2 -2844.787} C_VEL
LIN {X 0,Y 559.159,Z 42.833,A -85,B 0,C 180,E1 -2847.365,E2 -2847.365} C_VEL
LIN {X 0,Y 559.153,Z 42.83,A -85,B 0,C 180,E1 -2850.143,E2 -2850.143} C_VEL
LIN {X 0,Y 559.174,Z 42.832,A -85,B 0,C 180,E1 -2853.098,E2 -2853.098} C_VEL
LIN {X 0,Y 559.162,Z 42.829,A -85,B 0,C 180,E1 -2855.495,E2 -2855.495} C_VEL
LIN {X 0,Y 559.177,Z 42.836,A -85,B 0,C 180,E1 -2858.624,E2 -2858.624} C_VEL
LIN {X 0,Y 559.166,Z 42.831,A -85,B 0,C 180,E1 -2860.926,E2 -2860.926} C_VEL
LIN {X 0,Y 559.167,Z 42.83,A -85,B 0,C 180,E1 -2863.948,E2 -2863.948} C_VEL
LIN {X 0,Y 559.176,Z 42.833,A -85,B 0,C 180,E1 -2866.184,E2 -2866.184} C_VEL
LIN {X 0,Y 559.201,Z 42.823,A -85,B 0,C 180,E1 -2869.134,E2 -2869.134} C_VEL
LIN {X 0,Y 559.198,Z 42.832,A -85,B 0,C 180,E1 -2872.054,E2 -2872.054} C_VEL
LIN {X 0,Y 559.255,Z 42.817,A -85,B 0,C 180,E1 -2874.953,E2 -2874.953} C_VEL
LIN {X 0,Y 559.255,Z 42.825,A -85,B 0,C 180,E1 -2877.84,E2 -2877.84} C_VEL
LIN {X 0,Y 559.274,Z 42.814,A -85,B 0,C 180,E1 -2880.72,E2 -2880.72} C_VEL
LIN {X 0,Y 559.24,Z 42.819,A -85,B 0,C 180,E1 -2882.881,E2 -2882.881} C_VEL
LIN {X 0,Y 559.223,Z 42.828,A -85,B 0,C 180,E1 -2885.77,E2 -2885.77} C_VEL
LIN {X 0,Y 559.175,Z 42.827,A -85,B 0,C 180,E1 -2888.675,E2 -2888.675} C_VEL
LIN {X 0,Y 559.212,Z 42.829,A -85,B 0,C 180,E1 -2891.6,E2 -2891.6} C_VEL
LIN {X 0,Y 559.207,Z 42.823,A -85,B 0,C 180,E1 -2894.595,E2 -2894.595} C_VEL
LIN {X 0,Y 559.147,Z 42.834,A -85,B 0,C 180,E1 -2897.557,E2 -2897.557} C_VEL
LIN {X 0,Y 559.171,Z 42.828,A -85,B 0,C 180,E1 -2899.838,E2 -2899.838} C_VEL
LIN {X 0,Y 559.146,Z 42.83,A -85,B 0,C 180,E1 -2902.153,E2 -2902.153} C_VEL
LIN {X 0,Y 559.18,Z 42.83,A -85,B 0,C 180,E1 -2905.298,E2 -2905.298} C_VEL
LIN {X 0,Y 559.135,Z 42.832,A -85,B 0,C 180,E1 -2907.715,E2 -2907.715} C_VEL
LIN {X 0,Y 559.158,Z 42.83,A -85,B 0,C 180,E1 -2910.183,E2 -2910.183} C_VEL
LIN {X 0,Y 559.156,Z 42.838,A -85,B 0,C 180,E1 -2912.715,E2 -2912.715} C_VEL
LIN {X 0,Y 559.128,Z 42.833,A -85,B 0,C 180,E1 -2915.324,E2 -2915.324} C_VEL
LIN {X 0,Y 559.134,Z 42.834,A -85,B 0,C 180,E1 -2918.018,E2 -2918.018} C_VEL
LIN {X 0,Y 559.16,Z 42.832,A -85,B 0,C 180,E1 -2920.812,E2 -2920.812} C_VEL
LIN {X 0,Y 559.142,Z 42.833,A -85,B 0,C 180,E1 -2923.734,E2 -2923.734} C_VEL
LIN {X 0,Y 559.135,Z 42.833,A -85,B 0,C 180,E1 -2926.805,E2 -2926.805} C_VEL
LIN {X 0,Y 559.159,Z 42.829,A -85,B 0,C 180,E1 -2929.187,E2 -2929.187} C_VEL
LIN {X 0,Y 559.133,Z 42.841,A -85,B 0,C 180,E1 -2931.982,E2 -2931.982} C_VEL
LIN {X 0,Y 559.134,Z 42.832,A -85,B 0,C 180,E1 -2934.787,E2 -2934.787} C_VEL
LIN {X 0,Y 559.157,Z 42.832,A -85,B 0,C 180,E1 -2937.365,E2 -2937.365} C_VEL
LIN {X 0,Y 559.148,Z 42.834,A -85,B 0,C 180,E1 -2940.143,E2 -2940.143} C_VEL
LIN {X 0,Y 559.168,Z 42.831,A -85,B 0,C 180,E1 -2943.097,E2 -2943.097} C_VEL
LIN {X 0,Y 559.227,Z 42.994,A -85,B 0,C 180,E1 -2945.523,E2 -2945.523} C_VEL
LIN {X 0,Y 560.119,Z 48.557,A -85,B 0,C 180,E1 -2946.342,E2 -2946.342} C_VEL
LIN {X 0,Y 559.874,Z 66.54,A -85,B 0,C 180,E1 -2948.845,E2 -2948.845} C_VEL
LIN {X 0,Y 559.698,Z 86.06,A -85,B 0,C 180,E1 -2951.515,E2 -2951.515} C_VEL
LIN {X 0,Y 559.486,Z 106.91,A -85,B 0,C 180,E1 -2954.331,E2 -2954.331} C_VEL
LIN {X 0,Y 559.374,Z 117.901,A -85,B 0,C 180,E1 -2955.806,E2 -2955.806} C_VEL
LIN {X 0,Y 560.288,Z 125.82,A -85,B 0,C 180,E1 -2955.934,E2 -2955.934} C_VEL
LIN {X 0,Y 560.033,Z 226.632,A -85,B 0,C 180,E1 -2957.244,E2 -2957.244} C_VEL
LIN {X 0,Y 559.922,Z 239.946,A -85,B 0,C 180,E1 -2957.564,E2 -2957.564} C_VEL
LIN {X 0,Y 559.812,Z 252.157,A -85,B 0,C 180,E1 -2957.999,E2 -2957.999} C_VEL
LIN {X 0,Y 559.622,Z 263.894,A -85,B 0,C 180,E1 -2958.559,E2 -2958.559} C_VEL
LIN {X 0,Y 559.456,Z 276.103,A -85,B 0,C 180,E1 -2959.322,E2 -2959.322} C_VEL
LIN {X 0,Y 559.305,Z 286.587,A -85,B 0,C 180,E1 -2960.142,E2 -2960.142} C_VEL
LIN {X 0,Y 559.162,Z 295.112,A -85,B 0,C 180,E1 -2960.961,E2 -2960.961} C_VEL
LIN {X 0,Y 559.05,Z 302.959,A -85,B 0,C 180,E1 -2961.869,E2 -2961.869} C_VEL
LIN {X 0,Y 558.944,Z 310.621,A -85,B 0,C 180,E1 -2962.958,E2 -2962.958} C_VEL
LIN {X 0,Y 558.936,Z 317.679,A -85,B 0,C 180,E1 -2964.227,E2 -2964.227} C_VEL
LIN {X 0,Y 558.826,Z 322.372,A -85,B 0,C 180,E1 -2965.311,E2 -2965.311} C_VEL
LIN {X 0,Y 558.836,Z 325.958,A -85,B 0,C 180,E1 -2966.395,E2 -2966.395} C_VEL
LIN {X 0,Y 558.799,Z 327.807,A -85,B 0,C 180,E1 -2967.116,E2 -2967.116} C_VEL
LIN {X 0,Y 558.745,Z 330.182,A -85,B 0,C 180,E1 -2968.558,E2 -2968.558} C_VEL
LIN {X 0,Y 558.74,Z 331,A -85,B 0,C 180,E1 -2970,E2 -2970} C_VEL
LIN {X 0,Y 558.745,Z 330.184,A -85,B 0,C 180,E1 -2971.441,E2 -2971.441} C_VEL
LIN {X 0,Y 558.799,Z 327.81,A -85,B 0,C 180,E1 -2972.884,E2 -2972.884} C_VEL
LIN {X 0,Y 558.844,Z 324.895,A -85,B 0,C 180,E1 -2973.966,E2 -2973.966} C_VEL
LIN {X 0,Y 558.798,Z 320.948,A -85,B 0,C 180,E1 -2975.051,E2 -2975.051} C_VEL
LIN {X 0,Y 558.923,Z 315.867,A -85,B 0,C 180,E1 -2976.136,E2 -2976.136} C_VEL
LIN {X 0,Y 558.977,Z 309.466,A -85,B 0,C 180,E1 -2977.223,E2 -2977.223} C_VEL
LIN {X 0,Y 559.099,Z 301.477,A -85,B 0,C 180,E1 -2978.312,E2 -2978.312} C_VEL
LIN {X 0,Y 559.195,Z 293.332,A -85,B 0,C 180,E1 -2979.221,E2 -2979.221} C_VEL
LIN {X 0,Y 559.353,Z 283.359,A -85,B 0,C 180,E1 -2980.131,E2 -2980.131} C_VEL
LIN {X 0,Y 559.526,Z 272.282,A -85,B 0,C 180,E1 -2980.937,E2 -2980.937} C_VEL
LIN {X 0,Y 559.672,Z 260.272,A -85,B 0,C 180,E1 -2981.628,E2 -2981.628} C_VEL
LIN {X 0,Y 559.834,Z 247.521,A -85,B 0,C 180,E1 -2982.184,E2 -2982.184} C_VEL
LIN {X 0,Y 559.958,Z 234.964,A -85,B 0,C 180,E1 -2982.573,E2 -2982.573} C_VEL
LIN {X 0,Y 560.092,Z 222.267,A -85,B 0,C 180,E1 -2982.823,E2 -2982.823} C_VEL
LIN {X 0,Y 560.212,Z 123.805,A -85,B 0,C 180,E1 -2984.094,E2 -2984.094} C_VEL
LIN {X 0,Y 559.353,Z 117.795,A -85,B 0,C 180,E1 -2984.206,E2 -2984.206} C_VEL
LIN {X 0,Y 559.579,Z 96.415,A -85,B 0,C 180,E1 -2987.075,E2 -2987.075} C_VEL
LIN {X 0,Y 559.836,Z 74.823,A -85,B 0,C 180,E1 -2990.004,E2 -2990.004} C_VEL
LIN {X 0,Y 560.078,Z 52.531,A -85,B 0,C 180,E1 -2993.087,E2 -2993.087} C_VEL
LIN {X 0,Y 559.955,Z 46.931,A -85,B 0,C 180,E1 -2993.877,E2 -2993.877} C_VEL
LIN {X 0,Y 559.207,Z 42.832,A -85,B 0,C 180,E1 -2994.503,E2 -2994.503} C_VEL
LIN {X 0,Y 559.172,Z 42.832,A -85,B 0,C 180,E1 -2996.902,E2 -2996.902} C_VEL
LIN {X 0,Y 559.151,Z 42.834,A -85,B 0,C 180,E1 -2999.857,E2 -2999.857} C_VEL
LIN {X 0,Y 559.156,Z 42.832,A -85,B 0,C 180,E1 -3002.716,E2 -3002.716} C_VEL
LIN {X 0,Y 559.131,Z 42.833,A -85,B 0,C 180,E1 -3005.324,E2 -3005.324} C_VEL
LIN {X 0,Y 559.136,Z 42.839,A -85,B 0,C 180,E1 -3008.018,E2 -3008.018} C_VEL
LIN {X 0,Y 559.159,Z 42.829,A -85,B 0,C 180,E1 -3010.813,E2 -3010.813} C_VEL
LIN {X 0,Y 559.159,Z 42.837,A -85,B 0,C 180,E1 -3013.732,E2 -3013.732} C_VEL
LIN {X 0,Y 559.148,Z 42.83,A -85,B 0,C 180,E1 -3016.804,E2 -3016.804} C_VEL
LIN {X 0,Y 559.159,Z 42.833,A -85,B 0,C 180,E1 -3019.188,E2 -3019.188} C_VEL
LIN {X 0,Y 559.136,Z 42.832,A -85,B 0,C 180,E1 -3021.982,E2 -3021.982} C_VEL
LIN {X 0,Y 559.136,Z 42.834,A -85,B 0,C 180,E1 -3024.787,E2 -3024.787} C_VEL
LIN {X 0,Y 559.157,Z 42.835,A -85,B 0,C 180,E1 -3027.365,E2 -3027.365} C_VEL
LIN {X 0,Y 559.153,Z 42.828,A -85,B 0,C 180,E1 -3030.143,E2 -3030.143} C_VEL
LIN {X 0,Y 559.174,Z 42.832,A -85,B 0,C 180,E1 -3033.098,E2 -3033.098} C_VEL
LIN {X 0,Y 559.16,Z 42.83,A -85,B 0,C 180,E1 -3035.495,E2 -3035.495} C_VEL
LIN {X 0,Y 559.177,Z 42.834,A -85,B 0,C 180,E1 -3038.624,E2 -3038.624} C_VEL
LIN {X 0,Y 559.165,Z 42.832,A -85,B 0,C 180,E1 -3040.926,E2 -3040.926} C_VEL
LIN {X 0,Y 559.169,Z 42.828,A -85,B 0,C 180,E1 -3043.948,E2 -3043.948} C_VEL
LIN {X 0,Y 559.175,Z 42.833,A -85,B 0,C 180,E1 -3046.184,E2 -3046.184} C_VEL
LIN {X 0,Y 559.2,Z 42.823,A -85,B 0,C 180,E1 -3049.134,E2 -3049.134} C_VEL
LIN {X 0,Y 559.205,Z 42.831,A -85,B 0,C 180,E1 -3052.054,E2 -3052.054} C_VEL
LIN {X 0,Y 559.254,Z 42.817,A -85,B 0,C 180,E1 -3054.953,E2 -3054.953} C_VEL
LIN {X 0,Y 559.254,Z 42.825,A -85,B 0,C 180,E1 -3057.839,E2 -3057.839} C_VEL
LIN {X 0,Y 559.274,Z 42.815,A -85,B 0,C 180,E1 -3060.72,E2 -3060.72} C_VEL
LIN {X 0,Y 559.239,Z 42.818,A -85,B 0,C 180,E1 -3062.881,E2 -3062.881} C_VEL
LIN {X 0,Y 559.221,Z 42.828,A -85,B 0,C 180,E1 -3065.77,E2 -3065.77} C_VEL
LIN {X 0,Y 559.173,Z 42.826,A -85,B 0,C 180,E1 -3068.675,E2 -3068.675} C_VEL
LIN {X 0,Y 559.21,Z 42.828,A -85,B 0,C 180,E1 -3071.6,E2 -3071.6} C_VEL
LIN {X 0,Y 559.205,Z 42.823,A -85,B 0,C 180,E1 -3074.595,E2 -3074.595} C_VEL
LIN {X 0,Y 559.145,Z 42.833,A -85,B 0,C 180,E1 -3077.557,E2 -3077.557} C_VEL
LIN {X 0,Y 559.17,Z 42.828,A -85,B 0,C 180,E1 -3079.837,E2 -3079.837} C_VEL
LIN {X 0,Y 559.144,Z 42.831,A -85,B 0,C 180,E1 -3082.153,E2 -3082.153} C_VEL
LIN {X 0,Y 559.178,Z 42.829,A -85,B 0,C 180,E1 -3085.298,E2 -3085.298} C_VEL
LIN {X 0,Y 559.131,Z 42.832,A -85,B 0,C 180,E1 -3087.715,E2 -3087.715} C_VEL
LIN {X 0,Y 559.141,Z 42.832,A -85,B 0,C 180,E1 -3090.606,E2 -3090.606} C_VEL
LIN {X 0,Y 558.479,Z 42.916,A -85,B 0,C 180,E1 -3091.207,E2 -3091.207} C_VEL
LIN {X 0,Y 555.615,Z 43.274,A -85,B 0,C 180,E1 -3092.183,E2 -3092.183} C_VEL
LIN {X 0,Y 553.198,Z 43.574,A -85,B 0,C 180,E1 -3092.969,E2 -3092.969} C_VEL
LIN {X 0,Y 552.17,Z 43.699,A -85,B 0,C 180,E1 -3093.576,E2 -3093.576} C_VEL
LIN {X 0,Y 552.092,Z 43.71,A -85,B 0,C 180,E1 -3093.781,E2 -3093.781} C_VEL
LIN {X 0,Y 552.1,Z 43.711,A -85,B 0,C 180,E1 -3096.747,E2 -3096.747} C_VEL
LIN {X 0,Y 552.13,Z 43.705,A -85,B 0,C 180,E1 -3099.527,E2 -3099.527} C_VEL
LIN {X 0,Y 552.111,Z 43.712,A -85,B 0,C 180,E1 -3102.427,E2 -3102.427} C_VEL
LIN {X 0,Y 552.078,Z 43.715,A -85,B 0,C 180,E1 -3105.56,E2 -3105.56} C_VEL
LIN {X 0,Y 552.122,Z 43.706,A -85,B 0,C 180,E1 -3108.678,E2 -3108.678} C_VEL
LIN {X 0,Y 552.114,Z 43.711,A -85,B 0,C 180,E1 -3111.41,E2 -3111.41} C_VEL
LIN {X 0,Y 552.076,Z 43.715,A -85,B 0,C 180,E1 -3114.155,E2 -3114.155} C_VEL
LIN {X 0,Y 552.107,Z 43.71,A -85,B 0,C 180,E1 -3116.813,E2 -3116.813} C_VEL
LIN {X 0,Y 552.093,Z 43.719,A -85,B 0,C 180,E1 -3119.39,E2 -3119.39} C_VEL
LIN {X 0,Y 552.148,Z 43.805,A -85,B 0,C 180,E1 -3122.084,E2 -3122.084} C_VEL
LIN {X 0,Y 552.4,Z 48.062,A -85,B 0,C 180,E1 -3122.947,E2 -3122.947} C_VEL
LIN {X 0,Y 552.242,Z 61.553,A -85,B 0,C 180,E1 -3125.634,E2 -3125.634} C_VEL
LIN {X 0,Y 552.259,Z 62.08,A -85,B 0,C 180,E1 -3125.7,E2 -3125.7} C_VEL
LIN {X 0,Y 553.444,Z 69.057,A -85,B 0,C 180,E1 -3125.824,E2 -3125.824} C_VEL
LIN {X 0,Y 553.123,Z 167.674,A -85,B 0,C 180,E1 -3127.125,E2 -3127.125} C_VEL
LIN {X 0,Y 553.035,Z 180.729,A -85,B 0,C 180,E1 -3127.441,E2 -3127.441} C_VEL
LIN {X 0,Y 552.938,Z 191.717,A -85,B 0,C 180,E1 -3127.831,E2 -3127.831} C_VEL
LIN {X 0,Y 552.754,Z 203.035,A -85,B 0,C 180,E1 -3128.363,E2 -3128.363} C_VEL
LIN {X 0,Y 552.527,Z 214.234,A -85,B 0,C 180,E1 -3129.038,E2 -3129.038} C_VEL
LIN {X 0,Y 552.37,Z 224.396,A -85,B 0,C 180,E1 -3129.811,E2 -3129.811} C_VEL
LIN {X 0,Y 552.2,Z 233.672,A -85,B 0,C 180,E1 -3130.676,E2 -3130.676} C_VEL
LIN {X 0,Y 552.071,Z 242.105,A -85,B 0,C 180,E1 -3131.635,E2 -3131.635} C_VEL
LIN {X 0,Y 551.957,Z 250.025,A -85,B 0,C 180,E1 -3132.74,E2 -3132.74} C_VEL
LIN {X 0,Y 551.858,Z 255.766,A -85,B 0,C 180,E1 -3133.729,E2 -3133.729} C_VEL
LIN {X 0,Y 551.796,Z 261.07,A -85,B 0,C 180,E1 -3134.865,E2 -3134.865} C_VEL
LIN {X 0,Y 551.746,Z 265.136,A -85,B 0,C 180,E1 -3135.994,E2 -3135.994} C_VEL
LIN {X 0,Y 551.688,Z 267.209,A -85,B 0,C 180,E1 -3136.744,E2 -3136.744} C_VEL
LIN {X 0,Y 551.688,Z 268.848,A -85,B 0,C 180,E1 -3137.493,E2 -3137.493} C_VEL
LIN {X 0,Y 551.71,Z 270.668,A -85,B 0,C 180,E1 -3138.775,E2 -3138.775} C_VEL
LIN {X 0,Y 551.681,Z 271.209,A -85,B 0,C 180,E1 -3139.726,E2 -3139.726} C_VEL
LIN {X 0,Y 551.69,Z 270.773,A -85,B 0,C 180,E1 -3141.207,E2 -3141.207} C_VEL
LIN {X 0,Y 551.694,Z 269.924,A -85,B 0,C 180,E1 -3141.945,E2 -3141.945} C_VEL
LIN {X 0,Y 551.761,Z 267.026,A -85,B 0,C 180,E1 -3143.417,E2 -3143.417} C_VEL
LIN {X 0,Y 551.769,Z 263.723,A -85,B 0,C 180,E1 -3144.518,E2 -3144.518} C_VEL
LIN {X 0,Y 551.817,Z 259.362,A -85,B 0,C 180,E1 -3145.617,E2 -3145.617} C_VEL
LIN {X 0,Y 551.851,Z 253.836,A -85,B 0,C 180,E1 -3146.715,E2 -3146.715} C_VEL
LIN {X 0,Y 551.954,Z 246.944,A -85,B 0,C 180,E1 -3147.811,E2 -3147.811} C_VEL
LIN {X 0,Y 552.122,Z 238.333,A -85,B 0,C 180,E1 -3148.906,E2 -3148.906} C_VEL
LIN {X 0,Y 552.247,Z 229.555,A -85,B 0,C 180,E1 -3149.818,E2 -3149.818} C_VEL
LIN {X 0,Y 552.438,Z 218.73,A -85,B 0,C 180,E1 -3150.729,E2 -3150.729} C_VEL
LIN {X 0,Y 552.676,Z 207.779,A -85,B 0,C 180,E1 -3151.457,E2 -3151.457} C_VEL
LIN {X 0,Y 552.875,Z 195.555,A -85,B 0,C 180,E1 -3152.094,E2 -3152.094} C_VEL
LIN {X 0,Y 552.988,Z 183.939,A -85,B 0,C 180,E1 -3152.55,E2 -3152.55} C_VEL
LIN {X 0,Y 553.099,Z 171.319,A -85,B 0,C 180,E1 -3152.891,E2 -3152.891} C_VEL
LIN {X 0,Y 553.206,Z 153.53,A -85,B 0,C 180,E1 -3153.163,E2 -3153.163} C_VEL
LIN {X 0,Y 553.377,Z 68.119,A -85,B 0,C 180,E1 -3154.279,E2 -3154.279} C_VEL
LIN {X 0,Y 552.166,Z 61.837,A -85,B 0,C 180,E1 -3154.403,E2 -3154.403} C_VEL
LIN {X 0,Y 552.385,Z 50.886,A -85,B 0,C 180,E1 -3156.575,E2 -3156.575} C_VEL
LIN {X 0,Y 552.221,Z 43.989,A -85,B 0,C 180,E1 -3157.956,E2 -3157.956} C_VEL
LIN {X 0,Y 552.156,Z 43.708,A -85,B 0,C 180,E1 -3158.049,E2 -3158.049} C_VEL
LIN {X 0,Y 552.178,Z 43.698,A -85,B 0,C 180,E1 -3161.467,E2 -3161.467} C_VEL
LIN {X 0,Y 552.16,Z 43.708,A -85,B 0,C 180,E1 -3164.683,E2 -3164.683} C_VEL
LIN {X 0,Y 552.112,Z 43.707,A -85,B 0,C 180,E1 -3167.789,E2 -3167.789} C_VEL
LIN {X 0,Y 552.129,Z 43.709,A -85,B 0,C 180,E1 -3170.101,E2 -3170.101} C_VEL
LIN {X 0,Y 552.094,Z 43.715,A -85,B 0,C 180,E1 -3172.451,E2 -3172.451} C_VEL
LIN {X 0,Y 552.158,Z 43.701,A -85,B 0,C 180,E1 -3175.351,E2 -3175.351} C_VEL
LIN {X 0,Y 552.123,Z 43.714,A -85,B 0,C 180,E1 -3178.098,E2 -3178.098} C_VEL
LIN {X 0,Y 552.105,Z 43.709,A -85,B 0,C 180,E1 -3180.609,E2 -3180.609} C_VEL
LIN {X 0,Y 552.118,Z 43.706,A -85,B 0,C 180,E1 -3183.186,E2 -3183.186} C_VEL
LIN {X 0,Y 552.103,Z 43.716,A -85,B 0,C 180,E1 -3185.843,E2 -3185.843} C_VEL
LIN {X 0,Y 552.125,Z 43.706,A -85,B 0,C 180,E1 -3189.062,E2 -3189.062} C_VEL
LIN {X 0,Y 552.124,Z 43.712,A -85,B 0,C 180,E1 -3191.446,E2 -3191.446} C_VEL
LIN {X 0,Y 552.092,Z 43.709,A -85,B 0,C 180,E1 -3194.531,E2 -3194.531} C_VEL
LIN {X 0,Y 552.133,Z 43.71,A -85,B 0,C 180,E1 -3197.585,E2 -3197.585} C_VEL
LIN {X 0,Y 552.134,Z 43.704,A -85,B 0,C 180,E1 -3200.473,E2 -3200.473} C_VEL
LIN {X 0,Y 552.11,Z 43.714,A -85,B 0,C 180,E1 -3203.317,E2 -3203.317} C_VEL
LIN {X 0,Y 552.132,Z 43.704,A -85,B 0,C 180,E1 -3205.939,E2 -3205.939} C_VEL
LIN {X 0,Y 552.124,Z 43.708,A -85,B 0,C 180,E1 -3208.541,E2 -3208.541} C_VEL
LIN {X 0,Y 552.129,Z 43.706,A -85,B 0,C 180,E1 -3211.438,E2 -3211.438} C_VEL
LIN {X 0,Y 552.134,Z 43.707,A -85,B 0,C 180,E1 -3214.356,E2 -3214.356} C_VEL
LIN {X 0,Y 552.104,Z 43.716,A -85,B 0,C 180,E1 -3216.758,E2 -3216.758} C_VEL
LIN {X 0,Y 552.123,Z 43.707,A -85,B 0,C 180,E1 -3219.12,E2 -3219.12} C_VEL
LIN {X 0,Y 552.099,Z 43.708,A -85,B 0,C 180,E1 -3221.444,E2 -3221.444} C_VEL
LIN {X 0,Y 552.117,Z 43.707,A -85,B 0,C 180,E1 -3223.737,E2 -3223.737} C_VEL
LIN {X 0,Y 552.14,Z 43.707,A -85,B 0,C 180,E1 -3226.005,E2 -3226.005} C_VEL
LIN {X 0,Y 552.169,Z 43.7,A -85,B 0,C 180,E1 -3228.994,E2 -3228.994} C_VEL
LIN {X 0,Y 552.153,Z 43.708,A -85,B 0,C 180,E1 -3231.952,E2 -3231.952} C_VEL
LIN {X 0,Y 552.23,Z 43.692,A -85,B 0,C 180,E1 -3234.889,E2 -3234.889} C_VEL
LIN {X 0,Y 552.227,Z 43.7,A -85,B 0,C 180,E1 -3237.812,E2 -3237.812} C_VEL
LIN {X 0,Y 552.245,Z 43.69,A -85,B 0,C 180,E1 -3240.729,E2 -3240.729} C_VEL
LIN {X 0,Y 552.207,Z 43.695,A -85,B 0,C 180,E1 -3242.918,E2 -3242.918} C_VEL
LIN {X 0,Y 552.192,Z 43.703,A -85,B 0,C 180,E1 -3245.844,E2 -3245.844} C_VEL
LIN {X 0,Y 552.146,Z 43.703,A -85,B 0,C 180,E1 -3248.786,E2 -3248.786} C_VEL
LIN {X 0,Y 552.169,Z 43.704,A -85,B 0,C 180,E1 -3251.75,E2 -3251.75} C_VEL
LIN {X 0,Y 552.143,Z 43.704,A -85,B 0,C 180,E1 -3254.748,E2 -3254.748} C_VEL
LIN {X 0,Y 552.104,Z 43.709,A -85,B 0,C 180,E1 -3257.789,E2 -3257.789} C_VEL
LIN {X 0,Y 552.132,Z 43.704,A -85,B 0,C 180,E1 -3260.101,E2 -3260.101} C_VEL
LIN {X 0,Y 552.097,Z 43.71,A -85,B 0,C 180,E1 -3262.451,E2 -3262.451} C_VEL
LIN {X 0,Y 552.143,Z 43.706,A -85,B 0,C 180,E1 -3265.346,E2 -3265.346} C_VEL
LIN {X 0,Y 552.09,Z 43.71,A -85,B 0,C 180,E1 -3268.1,E2 -3268.1} C_VEL
LIN {X 0,Y 552.107,Z 43.714,A -85,B 0,C 180,E1 -3270.609,E2 -3270.609} C_VEL
LIN {X 0,Y 552.111,Z 43.709,A -85,B 0,C 180,E1 -3273.186,E2 -3273.186} C_VEL
LIN {X 0,Y 552.08,Z 43.711,A -85,B 0,C 180,E1 -3275.844,E2 -3275.844} C_VEL
LIN {X 0,Y 552.12,Z 43.713,A -85,B 0,C 180,E1 -3278.589,E2 -3278.589} C_VEL
LIN {X 0,Y 552.125,Z 43.705,A -85,B 0,C 180,E1 -3281.446,E2 -3281.446} C_VEL
LIN {X 0,Y 552.093,Z 43.714,A -85,B 0,C 180,E1 -3284.531,E2 -3284.531} C_VEL
LIN {X 0,Y 552.113,Z 43.708,A -85,B 0,C 180,E1 -3287.587,E2 -3287.587} C_VEL
LIN {X 0,Y 552.132,Z 43.707,A -85,B 0,C 180,E1 -3290.473,E2 -3290.473} C_VEL
LIN {X 0,Y 552.103,Z 43.709,A -85,B 0,C 180,E1 -3293.318,E2 -3293.318} C_VEL
LIN {X 0,Y 552.123,Z 43.713,A -85,B 0,C 180,E1 -3295.938,E2 -3295.938} C_VEL
LIN {X 0,Y 552.123,Z 43.705,A -85,B 0,C 180,E1 -3298.541,E2 -3298.541} C_VEL
LIN {X 0,Y 552.128,Z 43.712,A -85,B 0,C 180,E1 -3301.438,E2 -3301.438} C_VEL
LIN {X 0,Y 552.131,Z 43.707,A -85,B 0,C 180,E1 -3304.356,E2 -3304.356} C_VEL
LIN {X 0,Y 552.179,Z 43.864,A -85,B 0,C 180,E1 -3305.365,E2 -3305.365} C_VEL
LIN {X 0,Y 553.188,Z 50.059,A -85,B 0,C 180,E1 -3306.291,E2 -3306.291} C_VEL
LIN {X 0,Y 552.925,Z 68.99,A -85,B 0,C 180,E1 -3308.956,E2 -3308.956} C_VEL
LIN {X 0,Y 552.696,Z 89.875,A -85,B 0,C 180,E1 -3311.848,E2 -3311.848} C_VEL
LIN {X 0,Y 552.366,Z 112.342,A -85,B 0,C 180,E1 -3314.918,E2 -3314.918} C_VEL
LIN {X 0,Y 552.311,Z 117.502,A -85,B 0,C 180,E1 -3315.619,E2 -3315.619} C_VEL
LIN {X 0,Y 553.403,Z 125.638,A -85,B 0,C 180,E1 -3315.758,E2 -3315.758} C_VEL
LIN {X 0,Y 553.114,Z 226.231,A -85,B 0,C 180,E1 -3317.082,E2 -3317.082} C_VEL
LIN {X 0,Y 552.973,Z 239.551,A -85,B 0,C 180,E1 -3317.405,E2 -3317.405} C_VEL
LIN {X 0,Y 552.849,Z 251.757,A -85,B 0,C 180,E1 -3317.845,E2 -3317.845} C_VEL
LIN {X 0,Y 552.65,Z 262.675,A -85,B 0,C 180,E1 -3318.369,E2 -3318.369} C_VEL
LIN {X 0,Y 552.469,Z 274.416,A -85,B 0,C 180,E1 -3319.092,E2 -3319.092} C_VEL
LIN {X 0,Y 552.258,Z 285.123,A -85,B 0,C 180,E1 -3319.922,E2 -3319.922} C_VEL
LIN {X 0,Y 552.11,Z 294.777,A -85,B 0,C 180,E1 -3320.844,E2 -3320.844} C_VEL
LIN {X 0,Y 551.984,Z 302.693,A -85,B 0,C 180,E1 -3321.765,E2 -3321.765} C_VEL
LIN {X 0,Y 551.89,Z 310.428,A -85,B 0,C 180,E1 -3322.868,E2 -3322.868} C_VEL
LIN {X 0,Y 551.845,Z 317.562,A -85,B 0,C 180,E1 -3324.152,E2 -3324.152} C_VEL
LIN {X 0,Y 551.723,Z 322.303,A -85,B 0,C 180,E1 -3325.25,E2 -3325.25} C_VEL
LIN {X 0,Y 551.75,Z 325.932,A -85,B 0,C 180,E1 -3326.348,E2 -3326.348} C_VEL
LIN {X 0,Y 551.723,Z 327.795,A -85,B 0,C 180,E1 -3327.079,E2 -3327.079} C_VEL
LIN {X 0,Y 551.645,Z 330.179,A -85,B 0,C 180,E1 -3328.54,E2 -3328.54} C_VEL
LIN {X 0,Y 551.64,Z 331,A -85,B 0,C 180,E1 -3330,E2 -3330} C_VEL
LIN {X 0,Y 551.645,Z 330.181,A -85,B 0,C 180,E1 -3331.46,E2 -3331.46} C_VEL
LIN {X 0,Y 551.723,Z 327.799,A -85,B 0,C 180,E1 -3332.921,E2 -3332.921} C_VEL
LIN {X 0,Y 551.764,Z 324.858,A -85,B 0,C 180,E1 -3334.017,E2 -3334.017} C_VEL
LIN {X 0,Y 551.723,Z 320.861,A -85,B 0,C 180,E1 -3335.116,E2 -3335.116} C_VEL
LIN {X 0,Y 551.798,Z 315.036,A -85,B 0,C 180,E1 -3336.342,E2 -3336.342} C_VEL
LIN {X 0,Y 551.892,Z 308.014,A -85,B 0,C 180,E1 -3337.5,E2 -3337.5} C_VEL
LIN {X 0,Y 552.038,Z 299.694,A -85,B 0,C 180,E1 -3338.603,E2 -3338.603} C_VEL
LIN {X 0,Y 552.163,Z 291.166,A -85,B 0,C 180,E1 -3339.524,E2 -3339.524} C_VEL
LIN {X 0,Y 552.366,Z 280.637,A -85,B 0,C 180,E1 -3340.446,E2 -3340.446} C_VEL
LIN {X 0,Y 552.555,Z 268.643,A -85,B 0,C 180,E1 -3341.286,E2 -3341.286} C_VEL
LIN {X 0,Y 552.757,Z 256.883,A -85,B 0,C 180,E1 -3341.924,E2 -3341.924} C_VEL
LIN {X 0,Y 552.93,Z 244.502,A -85,B 0,C 180,E1 -3342.432,E2 -3342.432} C_VEL
LIN {X 0,Y 553.037,Z 231.801,A -85,B 0,C 180,E1 -3342.803,E2 -3342.803} C_VEL
LIN {X 0,Y 553.166,Z 218.54,A -85,B 0,C 180,E1 -3343.033,E2 -3343.033} C_VEL
LIN {X 0,Y 553.214,Z 123.733,A -85,B 0,C 180,E1 -3344.271,E2 -3344.271} C_VEL
LIN {X 0,Y 552.316,Z 117.347,A -85,B 0,C 180,E1 -3344.397,E2 -3344.397} C_VEL
LIN {X 0,Y 552.585,Z 96.454,A -85,B 0,C 180,E1 -3347.24,E2 -3347.24} C_VEL
LIN {X 0,Y 552.889,Z 74.475,A -85,B 0,C 180,E1 -3350.267,E2 -3350.267} C_VEL
LIN {X 0,Y 553.208,Z 51.216,A -85,B 0,C 180,E1 -3353.526,E2 -3353.526} C_VEL
LIN {X 0,Y 552.443,Z 45.141,A -85,B 0,C 180,E1 -3354.422,E2 -3354.422} C_VEL
LIN {X 0,Y 552.174,Z 43.707,A -85,B 0,C 180,E1 -3354.66,E2 -3354.66} C_VEL
LIN {X 0,Y 552.133,Z 43.707,A -85,B 0,C 180,E1 -3357.274,E2 -3357.274} C_VEL
LIN {X 0,Y 552.12,Z 43.712,A -85,B 0,C 180,E1 -3360.051,E2 -3360.051} C_VEL
LIN {X 0,Y 552.114,Z 43.708,A -85,B 0,C 180,E1 -3362.846,E2 -3362.846} C_VEL
LIN {X 0,Y 552.08,Z 43.713,A -85,B 0,C 180,E1 -3365.44,E2 -3365.44} C_VEL
LIN {X 0,Y 552.1,Z 43.717,A -85,B 0,C 180,E1 -3367.886,E2 -3367.886} C_VEL
LIN {X 0,Y 552.112,Z 43.708,A -85,B 0,C 180,E1 -3370.481,E2 -3370.481} C_VEL
LIN {X 0,Y 552.123,Z 43.71,A -85,B 0,C 180,E1 -3373.485,E2 -3373.485} C_VEL
LIN {X 0,Y 552.11,Z 43.706,A -85,B 0,C 180,E1 -3376.576,E2 -3376.576} C_VEL
LIN {X 0,Y 552.112,Z 43.713,A -85,B 0,C 180,E1 -3379.519,E2 -3379.519} C_VEL
LIN {X 0,Y 552.096,Z 43.708,A -85,B 0,C 180,E1 -3382.336,E2 -3382.336} C_VEL
LIN {X 0,Y 552.087,Z 43.715,A -85,B 0,C 180,E1 -3385.051,E2 -3385.051} C_VEL
LIN {X 0,Y 552.118,Z 43.708,A -85,B 0,C 180,E1 -3387.681,E2 -3387.681} C_VEL
LIN {X 0,Y 552.116,Z 43.705,A -85,B 0,C 180,E1 -3390.235,E2 -3390.235} C_VEL
LIN {X 0,Y 552.143,Z 43.71,A -85,B 0,C 180,E1 -3393,E2 -3393} C_VEL
LIN {X 0,Y 552.118,Z 43.71,A -85,B 0,C 180,E1 -3395.161,E2 -3395.161} C_VEL
LIN {X 0,Y 552.131,Z 43.707,A -85,B 0,C 180,E1 -3398.337,E2 -3398.337} C_VEL
LIN {X 0,Y 552.155,Z 43.709,A -85,B 0,C 180,E1 -3400.674,E2 -3400.674} C_VEL
LIN {X 0,Y 552.119,Z 43.705,A -85,B 0,C 180,E1 -3403.737,E2 -3403.737} C_VEL
LIN {X 0,Y 552.139,Z 43.707,A -85,B 0,C 180,E1 -3406.004,E2 -3406.004} C_VEL
LIN {X 0,Y 552.168,Z 43.7,A -85,B 0,C 180,E1 -3408.993,E2 -3408.993} C_VEL
LIN {X 0,Y 552.16,Z 43.707,A -85,B 0,C 180,E1 -3411.951,E2 -3411.951} C_VEL
LIN {X 0,Y 552.229,Z 43.692,A -85,B 0,C 180,E1 -3414.889,E2 -3414.889} C_VEL
LIN {X 0,Y 552.226,Z 43.7,A -85,B 0,C 180,E1 -3417.812,E2 -3417.812} C_VEL
LIN {X 0,Y 552.244,Z 43.69,A -85,B 0,C 180,E1 -3420.729,E2 -3420.729} C_VEL
LIN {X 0,Y 552.206,Z 43.694,A -85,B 0,C 180,E1 -3422.918,E2 -3422.918} C_VEL
LIN {X 0,Y 552.19,Z 43.702,A -85,B 0,C 180,E1 -3425.844,E2 -3425.844} C_VEL
LIN {X 0,Y 552.144,Z 43.702,A -85,B 0,C 180,E1 -3428.786,E2 -3428.786} C_VEL
LIN {X 0,Y 552.168,Z 43.703,A -85,B 0,C 180,E1 -3431.75,E2 -3431.75} C_VEL
LIN {X 0,Y 552.141,Z 43.704,A -85,B 0,C 180,E1 -3434.748,E2 -3434.748} C_VEL
LIN {X 0,Y 552.102,Z 43.708,A -85,B 0,C 180,E1 -3437.789,E2 -3437.789} C_VEL
LIN {X 0,Y 552.13,Z 43.704,A -85,B 0,C 180,E1 -3440.101,E2 -3440.101} C_VEL
LIN {X 0,Y 552.095,Z 43.711,A -85,B 0,C 180,E1 -3442.451,E2 -3442.451} C_VEL
LIN {X 0,Y 552.141,Z 43.705,A -85,B 0,C 180,E1 -3445.346,E2 -3445.346} C_VEL
LIN {X 0,Y 552.081,Z 43.712,A -85,B 0,C 180,E1 -3448.1,E2 -3448.1} C_VEL
LIN {X 0,Y 552.104,Z 43.715,A -85,B 0,C 180,E1 -3450.609,E2 -3450.609} C_VEL
LIN {X 0,Y 552.11,Z 43.707,A -85,B 0,C 180,E1 -3453.186,E2 -3453.186} C_VEL
LIN {X 0,Y 552.092,Z 43.71,A -85,B 0,C 180,E1 -3453.781,E2 -3453.781} C_VEL
LIN {X 0,Y 551.45,Z 43.797,A -85,B 0,C 180,E1 -3454.39,E2 -3454.39} C_VEL
LIN {X 0,Y 548.634,Z 44.147,A -85,B 0,C 180,E1 -3455.378,E2 -3455.378} C_VEL
LIN {X 0,Y 546.224,Z 44.447,A -85,B 0,C 180,E1 -3456.173,E2 -3456.173} C_VEL
LIN {X 0,Y 545.16,Z 44.575,A -85,B 0,C 180,E1 -3456.787,E2 -3456.787} C_VEL
LIN {X 0,Y 545.059,Z 44.586,A -85,B 0,C 180,E1 -3456.995,E2 -3456.995} C_VEL
LIN {X 0,Y 545.067,Z 44.59,A -85,B 0,C 180,E1 -3460.143,E2 -3460.143} C_VEL
LIN {X 0,Y 545.047,Z 44.588,A -85,B 0,C 180,E1 -3463.11,E2 -3463.11} C_VEL
LIN {X 0,Y 545.047,Z 44.592,A -85,B 0,C 180,E1 -3466.227,E2 -3466.227} C_VEL
LIN {X 0,Y 545.082,Z 44.583,A -85,B 0,C 180,E1 -3468.885,E2 -3468.885} C_VEL
LIN {X 0,Y 545.045,Z 44.595,A -85,B 0,C 180,E1 -3471.865,E2 -3471.865} C_VEL
LIN {X 0,Y 545.031,Z 44.59,A -85,B 0,C 180,E1 -3474.531,E2 -3474.531} C_VEL
LIN {X 0,Y 545.065,Z 44.592,A -85,B 0,C 180,E1 -3477.211,E2 -3477.211} C_VEL
LIN {X 0,Y 545.063,Z 44.592,A -85,B 0,C 180,E1 -3479.81,E2 -3479.81} C_VEL
LIN {X 0,Y 545.109,Z 44.684,A -85,B 0,C 180,E1 -3481.98,E2 -3481.98} C_VEL
LIN {X 0,Y 545.452,Z 48.471,A -85,B 0,C 180,E1 -3482.754,E2 -3482.754} C_VEL
LIN {X 0,Y 545.279,Z 62.447,A -85,B 0,C 180,E1 -3485.512,E2 -3485.512} C_VEL
LIN {X 0,Y 546.527,Z 68.583,A -85,B 0,C 180,E1 -3485.629,E2 -3485.629} C_VEL
LIN {X 0,Y 546.222,Z 168.558,A -85,B 0,C 180,E1 -3486.969,E2 -3486.969} C_VEL
LIN {X 0,Y 546.113,Z 182.231,A -85,B 0,C 180,E1 -3487.314,E2 -3487.314} C_VEL
LIN {X 0,Y 545.977,Z 194.592,A -85,B 0,C 180,E1 -3487.778,E2 -3487.778} C_VEL
LIN {X 0,Y 545.755,Z 206.24,A -85,B 0,C 180,E1 -3488.369,E2 -3488.369} C_VEL
LIN {X 0,Y 545.494,Z 218.138,A -85,B 0,C 180,E1 -3489.15,E2 -3489.15} C_VEL
LIN {X 0,Y 545.353,Z 228.154,A -85,B 0,C 180,E1 -3489.976,E2 -3489.976} C_VEL
LIN {X 0,Y 545.189,Z 236.456,A -85,B 0,C 180,E1 -3490.809,E2 -3490.809} C_VEL
LIN {X 0,Y 544.989,Z 244.447,A -85,B 0,C 180,E1 -3491.777,E2 -3491.777} C_VEL
LIN {X 0,Y 544.887,Z 252.179,A -85,B 0,C 180,E1 -3492.936,E2 -3492.936} C_VEL
LIN {X 0,Y 544.776,Z 257.401,A -85,B 0,C 180,E1 -3493.897,E2 -3493.897} C_VEL
LIN {X 0,Y 544.725,Z 262.411,A -85,B 0,C 180,E1 -3495.046,E2 -3495.046} C_VEL
LIN {X 0,Y 544.659,Z 266.23,A -85,B 0,C 180,E1 -3496.189,E2 -3496.189} C_VEL
LIN {X 0,Y 544.598,Z 268.977,A -85,B 0,C 180,E1 -3497.327,E2 -3497.327} C_VEL
LIN {X 0,Y 544.62,Z 271.028,A -85,B 0,C 180,E1 -3498.735,E2 -3498.735} C_VEL
LIN {X 0,Y 544.592,Z 271.565,A -85,B 0,C 180,E1 -3499.591,E2 -3499.591} C_VEL
LIN {X 0,Y 544.603,Z 271.244,A -85,B 0,C 180,E1 -3501.091,E2 -3501.091} C_VEL
LIN {X 0,Y 544.612,Z 270.497,A -85,B 0,C 180,E1 -3501.839,E2 -3501.839} C_VEL
LIN {X 0,Y 544.62,Z 269.31,A -85,B 0,C 180,E1 -3502.586,E2 -3502.586} C_VEL
LIN {X 0,Y 544.68,Z 267.365,A -85,B 0,C 180,E1 -3503.479,E2 -3503.479} C_VEL
LIN {X 0,Y 544.665,Z 263.263,A -85,B 0,C 180,E1 -3504.818,E2 -3504.818} C_VEL
LIN {X 0,Y 544.779,Z 258.647,A -85,B 0,C 180,E1 -3505.931,E2 -3505.931} C_VEL
LIN {X 0,Y 544.834,Z 251.73,A -85,B 0,C 180,E1 -3507.227,E2 -3507.227} C_VEL
LIN {X 0,Y 544.989,Z 244.25,A -85,B 0,C 180,E1 -3508.337,E2 -3508.337} C_VEL
LIN {X 0,Y 545.192,Z 236.609,A -85,B 0,C 180,E1 -3509.261,E2 -3509.261} C_VEL
LIN {X 0,Y 545.296,Z 226.299,A -85,B 0,C 180,E1 -3510.277,E2 -3510.277} C_VEL
LIN {X 0,Y 545.543,Z 215.799,A -85,B 0,C 180,E1 -3511.107,E2 -3511.107} C_VEL
LIN {X 0,Y 545.735,Z 205.674,A -85,B 0,C 180,E1 -3511.753,E2 -3511.753} C_VEL
LIN {X 0,Y 545.96,Z 193.627,A -85,B 0,C 180,E1 -3512.352,E2 -3512.352} C_VEL
LIN {X 0,Y 546.096,Z 181.035,A -85,B 0,C 180,E1 -3512.812,E2 -3512.812} C_VEL
LIN {X 0,Y 546.242,Z 167.805,A -85,B 0,C 180,E1 -3513.135,E2 -3513.135} C_VEL
LIN {X 0,Y 546.477,Z 68.68,A -85,B 0,C 180,E1 -3514.46,E2 -3514.46} C_VEL
LIN {X 0,Y 545.199,Z 62.126,A -85,B 0,C 180,E1 -3514.598,E2 -3514.598} C_VEL
LIN {X 0,Y 545.413,Z 50.736,A -85,B 0,C 180,E1 -3516.871,E2 -3516.871} C_VEL
LIN {X 0,Y 545.171,Z 44.861,A -85,B 0,C 180,E1 -3518.059,E2 -3518.059} C_VEL
LIN {X 0,Y 545.127,Z 44.584,A -85,B 0,C 180,E1 -3518.153,E2 -3518.153} C_VEL
LIN {X 0,Y 545.138,Z 44.575,A -85,B 0,C 180,E1 -3521.535,E2 -3521.535} C_VEL
LIN {X 0,Y 545.106,Z 44.585,A -85,B 0,C 180,E1 -3524.767,E2 -3524.767} C_VEL
LIN {X 0,Y 545.095,Z 44.58,A -85,B 0,C 180,E1 -3527.428,E2 -3527.428} C_VEL
LIN {X 0,Y 545.095,Z 44.59,A -85,B 0,C 180,E1 -3530.372,E2 -3530.372} C_VEL
LIN {X 0,Y 545.081,Z 44.583,A -85,B 0,C 180,E1 -3533.56,E2 -3533.56} C_VEL
LIN {X 0,Y 545.082,Z 44.589,A -85,B 0,C 180,E1 -3536.001,E2 -3536.001} C_VEL
LIN {X 0,Y 545.092,Z 44.582,A -85,B 0,C 180,E1 -3538.748,E2 -3538.748} C_VEL
LIN {X 0,Y 545.06,Z 44.59,A -85,B 0,C 180,E1 -3541.679,E2 -3541.679} C_VEL
LIN {X 0,Y 545.081,Z 44.583,A -85,B 0,C 180,E1 -3544.564,E2 -3544.564} C_VEL
LIN {X 0,Y 545.04,Z 44.59,A -85,B 0,C 180,E1 -3547.304,E2 -3547.304} C_VEL
LIN {X 0,Y 545.069,Z 44.586,A -85,B 0,C 180,E1 -3550.143,E2 -3550.143} C_VEL
LIN {X 0,Y 545.081,Z 44.585,A -85,B 0,C 180,E1 -3553.107,E2 -3553.107} C_VEL
LIN {X 0,Y 545.052,Z 44.586,A -85,B 0,C 180,E1 -3556.227,E2 -3556.227} C_VEL
LIN {X 0,Y 545.085,Z 44.585,A -85,B 0,C 180,E1 -3558.886,E2 -3558.886} C_VEL
LIN {X 0,Y 545.084,Z 44.585,A -85,B 0,C 180,E1 -3560.819,E2 -3560.819} C_VEL
LIN {X 0,Y 545.046,Z 44.589,A -85,B 0,C 180,E1 -3563.62,E2 -3563.62} C_VEL
LIN {X 0,Y 545.07,Z 44.584,A -85,B 0,C 180,E1 -3566.328,E2 -3566.328} C_VEL
LIN {X 0,Y 545.07,Z 44.593,A -85,B 0,C 180,E1 -3568.952,E2 -3568.952} C_VEL
LIN {X 0,Y 545.106,Z 44.58,A -85,B 0,C 180,E1 -3571.508,E2 -3571.508} C_VEL
LIN {X 0,Y 545.099,Z 44.585,A -85,B 0,C 180,E1 -3574.492,E2 -3574.492} C_VEL
LIN {X 0,Y 545.043,Z 44.589,A -85,B 0,C 180,E1 -3577.243,E2 -3577.243} C_VEL
LIN {X 0,Y 545.122,Z 44.584,A -85,B 0,C 180,E1 -3580.415,E2 -3580.415} C_VEL
LIN {X 0,Y 545.069,Z 44.584,A -85,B 0,C 180,E1 -3583.521,E2 -3583.521} C_VEL
LIN {X 0,Y 545.1,Z 44.582,A -85,B 0,C 180,E1 -3585.82,E2 -3585.82} C_VEL
LIN {X 0,Y 545.124,Z 44.578,A -85,B 0,C 180,E1 -3588.85,E2 -3588.85} C_VEL
LIN {X 0,Y 545.102,Z 44.584,A -85,B 0,C 180,E1 -3591.847,E2 -3591.847} C_VEL
LIN {X 0,Y 545.173,Z 44.58,A -85,B 0,C 180,E1 -3594.081,E2 -3594.081} C_VEL
LIN {X 0,Y 545.173,Z 44.571,A -85,B 0,C 180,E1 -3597.044,E2 -3597.044} C_VEL
LIN {X 0,Y 545.207,Z 44.574,A -85,B 0,C 180,E1 -3600,E2 -3600} C_VEL
LIN {X 0,Y 545.174,Z 44.571,A -85,B 0,C 180,E1 -3602.956,E2 -3602.956} C_VEL
LIN {X 0,Y 545.141,Z 44.58,A -85,B 0,C 180,E1 -3605.92,E2 -3605.92} C_VEL
LIN {X 0,Y 545.103,Z 44.581,A -85,B 0,C 180,E1 -3608.153,E2 -3608.153} C_VEL
LIN {X 0,Y 545.142,Z 44.582,A -85,B 0,C 180,E1 -3611.535,E2 -3611.535} C_VEL
LIN {X 0,Y 545.11,Z 44.581,A -85,B 0,C 180,E1 -3614.767,E2 -3614.767} C_VEL
LIN {X 0,Y 545.082,Z 44.588,A -85,B 0,C 180,E1 -3617.422,E2 -3617.422} C_VEL
LIN {X 0,Y 545.098,Z 44.581,A -85,B 0,C 180,E1 -3620.372,E2 -3620.372} C_VEL
LIN {X 0,Y 545.084,Z 44.584,A -85,B 0,C 180,E1 -3623.559,E2 -3623.559} C_VEL
LIN {X 0,Y 545.08,Z 44.582,A -85,B 0,C 180,E1 -3626.001,E2 -3626.001} C_VEL
LIN {X 0,Y 545.092,Z 44.589,A -85,B 0,C 180,E1 -3628.747,E2 -3628.747} C_VEL
LIN {X 0,Y 545.063,Z 44.584,A -85,B 0,C 180,E1 -3631.679,E2 -3631.679} C_VEL
LIN {X 0,Y 545.063,Z 44.593,A -85,B 0,C 180,E1 -3634.565,E2 -3634.565} C_VEL
LIN {X 0,Y 545.035,Z 44.588,A -85,B 0,C 180,E1 -3637.304,E2 -3637.304} C_VEL
LIN {X 0,Y 545.069,Z 44.589,A -85,B 0,C 180,E1 -3640.143,E2 -3640.143} C_VEL
LIN {X 0,Y 545.083,Z 44.582,A -85,B 0,C 180,E1 -3643.106,E2 -3643.106} C_VEL
LIN {X 0,Y 545.049,Z 44.595,A -85,B 0,C 180,E1 -3646.227,E2 -3646.227} C_VEL
LIN {X 0,Y 545.085,Z 44.582,A -85,B 0,C 180,E1 -3648.885,E2 -3648.885} C_VEL
LIN {X 0,Y 545.051,Z 44.593,A -85,B 0,C 180,E1 -3651.864,E2 -3651.864} C_VEL
LIN {X 0,Y 545.035,Z 44.589,A -85,B 0,C 180,E1 -3654.531,E2 -3654.531} C_VEL
LIN {X 0,Y 545.069,Z 44.585,A -85,B 0,C 180,E1 -3657.211,E2 -3657.211} C_VEL
LIN {X 0,Y 545.065,Z 44.593,A -85,B 0,C 180,E1 -3659.81,E2 -3659.81} C_VEL
LIN {X 0,Y 545.081,Z 44.585,A -85,B 0,C 180,E1 -3662.343,E2 -3662.343} C_VEL
LIN {X 0,Y 545.123,Z 44.721,A -85,B 0,C 180,E1 -3665.202,E2 -3665.202} C_VEL
LIN {X 0,Y 546.269,Z 51.697,A -85,B 0,C 180,E1 -3666.259,E2 -3666.259} C_VEL
LIN {X 0,Y 545.931,Z 72.813,A -85,B 0,C 180,E1 -3669.266,E2 -3669.266} C_VEL
LIN {X 0,Y 545.611,Z 94.157,A -85,B 0,C 180,E1 -3672.257,E2 -3672.257} C_VEL
LIN {X 0,Y 545.29,Z 115.155,A -85,B 0,C 180,E1 -3675.16,E2 -3675.16} C_VEL
LIN {X 0,Y 545.28,Z 117.108,A -85,B 0,C 180,E1 -3675.429,E2 -3675.429} C_VEL
LIN {X 0,Y 546.524,Z 126.72,A -85,B 0,C 180,E1 -3675.594,E2 -3675.594} C_VEL
LIN {X 0,Y 546.197,Z 225.829,A -85,B 0,C 180,E1 -3676.916,E2 -3676.916} C_VEL
LIN {X 0,Y 546.022,Z 239.155,A -85,B 0,C 180,E1 -3677.242,E2 -3677.242} C_VEL
LIN {X 0,Y 545.889,Z 251.365,A -85,B 0,C 180,E1 -3677.688,E2 -3677.688} C_VEL
LIN {X 0,Y 545.652,Z 262.783,A -85,B 0,C 180,E1 -3678.244,E2 -3678.244} C_VEL
LIN {X 0,Y 545.47,Z 274.028,A -85,B 0,C 180,E1 -3678.951,E2 -3678.951} C_VEL
LIN {X 0,Y 545.244,Z 284.736,A -85,B 0,C 180,E1 -3679.791,E2 -3679.791} C_VEL
LIN {X 0,Y 545.065,Z 294.39,A -85,B 0,C 180,E1 -3680.725,E2 -3680.725} C_VEL
LIN {X 0,Y 544.934,Z 302.308,A -85,B 0,C 180,E1 -3681.657,E2 -3681.657} C_VEL
LIN {X 0,Y 544.798,Z 310.043,A -85,B 0,C 180,E1 -3682.774,E2 -3682.774} C_VEL
LIN {X 0,Y 544.755,Z 317.177,A -85,B 0,C 180,E1 -3684.076,E2 -3684.076} C_VEL
LIN {X 0,Y 544.627,Z 321.919,A -85,B 0,C 180,E1 -3685.188,E2 -3685.188} C_VEL
LIN {X 0,Y 544.669,Z 325.549,A -85,B 0,C 180,E1 -3686.301,E2 -3686.301} C_VEL
LIN {X 0,Y 544.65,Z 327.42,A -85,B 0,C 180,E1 -3687.041,E2 -3687.041} C_VEL
LIN {X 0,Y 544.552,Z 329.819,A -85,B 0,C 180,E1 -3688.521,E2 -3688.521} C_VEL
LIN {X 0,Y 544.55,Z 330.43,A -85,B 0,C 180,E1 -3689.26,E2 -3689.26} C_VEL
LIN {X 0,Y 544.55,Z 330.647,A -85,B 0,C 180,E1 -3690,E2 -3690} C_VEL
LIN {X 0,Y 544.55,Z 330.43,A -85,B 0,C 180,E1 -3690.739,E2 -3690.739} C_VEL
LIN {X 0,Y 544.571,Z 328.82,A -85,B 0,C 180,E1 -3692.219,E2 -3692.219} C_VEL
LIN {X 0,Y 544.65,Z 327.42,A -85,B 0,C 180,E1 -3692.959,E2 -3692.959} C_VEL
LIN {X 0,Y 544.684,Z 324.47,A -85,B 0,C 180,E1 -3694.069,E2 -3694.069} C_VEL
LIN {X 0,Y 544.653,Z 320.473,A -85,B 0,C 180,E1 -3695.182,E2 -3695.182} C_VEL
LIN {X 0,Y 544.7,Z 315.192,A -85,B 0,C 180,E1 -3696.324,E2 -3696.324} C_VEL
LIN {X 0,Y 544.822,Z 308.865,A -85,B 0,C 180,E1 -3697.412,E2 -3697.412} C_VEL
LIN {X 0,Y 544.95,Z 300.797,A -85,B 0,C 180,E1 -3698.529,E2 -3698.529} C_VEL
LIN {X 0,Y 545.083,Z 292.578,A -85,B 0,C 180,E1 -3699.462,E2 -3699.462} C_VEL
LIN {X 0,Y 545.32,Z 282.563,A -85,B 0,C 180,E1 -3700.395,E2 -3700.395} C_VEL
LIN {X 0,Y 545.486,Z 271.686,A -85,B 0,C 180,E1 -3701.209,E2 -3701.209} C_VEL
LIN {X 0,Y 545.704,Z 260.185,A -85,B 0,C 180,E1 -3701.892,E2 -3701.892} C_VEL
LIN {X 0,Y 545.898,Z 247.922,A -85,B 0,C 180,E1 -3702.453,E2 -3702.453} C_VEL
LIN {X 0,Y 546.085,Z 235.058,A -85,B 0,C 180,E1 -3702.874,E2 -3702.874} C_VEL
LIN {X 0,Y 546.225,Z 222.926,A -85,B 0,C 180,E1 -3703.131,E2 -3703.131} C_VEL
LIN {X 0,Y 546.372,Z 124.736,A -85,B 0,C 180,E1 -3704.435,E2 -3704.435} C_VEL
LIN {X 0,Y 545.255,Z 116.992,A -85,B 0,C 180,E1 -3704.581,E2 -3704.581} C_VEL
LIN {X 0,Y 545.574,Z 96.008,A -85,B 0,C 180,E1 -3707.476,E2 -3707.476} C_VEL
LIN {X 0,Y 545.916,Z 75.486,A -85,B 0,C 180,E1 -3710.34,E2 -3710.34} C_VEL
LIN {X 0,Y 546.298,Z 51.589,A -85,B 0,C 180,E1 -3713.736,E2 -3713.736} C_VEL
LIN {X 0,Y 545.1,Z 44.587,A -85,B 0,C 180,E1 -3714.824,E2 -3714.824} C_VEL
LIN {X 0,Y 545.084,Z 44.586,A -85,B 0,C 180,E1 -3717.656,E2 -3717.656} C_VEL
LIN {X 0,Y 545.081,Z 44.591,A -85,B 0,C 180,E1 -3720.246,E2 -3720.246} C_VEL
LIN {X 0,Y 545.077,Z 44.584,A -85,B 0,C 180,E1 -3723.061,E2 -3723.061} C_VEL
LIN {X 0,Y 545.037,Z 44.592,A -85,B 0,C 180,E1 -3725.673,E2 -3725.673} C_VEL
LIN {X 0,Y 545.055,Z 44.589,A -85,B 0,C 180,E1 -3728.237,E2 -3728.237} C_VEL
LIN {X 0,Y 545.084,Z 44.584,A -85,B 0,C 180,E1 -3730.473,E2 -3730.473} C_VEL
LIN {X 0,Y 545.082,Z 44.583,A -85,B 0,C 180,E1 -3733.107,E2 -3733.107} C_VEL
LIN {X 0,Y 545.052,Z 44.587,A -85,B 0,C 180,E1 -3736.226,E2 -3736.226} C_VEL
LIN {X 0,Y 545.085,Z 44.583,A -85,B 0,C 180,E1 -3738.885,E2 -3738.885} C_VEL
LIN {X 0,Y 545.084,Z 44.582,A -85,B 0,C 180,E1 -3740.818,E2 -3740.818} C_VEL
LIN {X 0,Y 545.046,Z 44.591,A -85,B 0,C 180,E1 -3743.62,E2 -3743.62} C_VEL
LIN {X 0,Y 545.054,Z 44.585,A -85,B 0,C 180,E1 -3746.327,E2 -3746.327} C_VEL
LIN {X 0,Y 545.071,Z 44.591,A -85,B 0,C 180,E1 -3748.952,E2 -3748.952} C_VEL
LIN {X 0,Y 545.106,Z 44.582,A -85,B 0,C 180,E1 -3751.508,E2 -3751.508} C_VEL
LIN {X 0,Y 545.099,Z 44.583,A -85,B 0,C 180,E1 -3754.491,E2 -3754.491} C_VEL
LIN {X 0,Y 545.041,Z 44.589,A -85,B 0,C 180,E1 -3757.242,E2 -3757.242} C_VEL
LIN {X 0,Y 545.121,Z 44.583,A -85,B 0,C 180,E1 -3760.415,E2 -3760.415} C_VEL
LIN {X 0,Y 545.07,Z 44.582,A -85,B 0,C 180,E1 -3763.521,E2 -3763.521} C_VEL
LIN {X 0,Y 545.099,Z 44.582,A -85,B 0,C 180,E1 -3765.82,E2 -3765.82} C_VEL
LIN {X 0,Y 545.123,Z 44.578,A -85,B 0,C 180,E1 -3768.849,E2 -3768.849} C_VEL
LIN {X 0,Y 545.131,Z 44.581,A -85,B 0,C 180,E1 -3771.847,E2 -3771.847} C_VEL
LIN {X 0,Y 545.206,Z 44.567,A -85,B 0,C 180,E1 -3774.823,E2 -3774.823} C_VEL
LIN {X 0,Y 545.198,Z 44.575,A -85,B 0,C 180,E1 -3777.784,E2 -3777.784} C_VEL
LIN {X 0,Y 545.215,Z 44.566,A -85,B 0,C 180,E1 -3780.738,E2 -3780.738} C_VEL
LIN {X 0,Y 545.173,Z 44.571,A -85,B 0,C 180,E1 -3782.956,E2 -3782.956} C_VEL
LIN {X 0,Y 545.14,Z 44.58,A -85,B 0,C 180,E1 -3785.92,E2 -3785.92} C_VEL
LIN {X 0,Y 545.102,Z 44.579,A -85,B 0,C 180,E1 -3788.153,E2 -3788.153} C_VEL
LIN {X 0,Y 545.141,Z 44.581,A -85,B 0,C 180,E1 -3791.534,E2 -3791.534} C_VEL
LIN {X 0,Y 545.108,Z 44.58,A -85,B 0,C 180,E1 -3794.767,E2 -3794.767} C_VEL
LIN {X 0,Y 545.08,Z 44.586,A -85,B 0,C 180,E1 -3797.422,E2 -3797.422} C_VEL
LIN {X 0,Y 545.096,Z 44.582,A -85,B 0,C 180,E1 -3800.372,E2 -3800.372} C_VEL
LIN {X 0,Y 545.082,Z 44.583,A -85,B 0,C 180,E1 -3803.559,E2 -3803.559} C_VEL
LIN {X 0,Y 545.078,Z 44.584,A -85,B 0,C 180,E1 -3806.001,E2 -3806.001} C_VEL
LIN {X 0,Y 545.072,Z 44.591,A -85,B 0,C 180,E1 -3808.744,E2 -3808.744} C_VEL
LIN {X 0,Y 545.061,Z 44.585,A -85,B 0,C 180,E1 -3811.679,E2 -3811.679} C_VEL
LIN {X 0,Y 545.059,Z 44.592,A -85,B 0,C 180,E1 -3814.565,E2 -3814.565} C_VEL
LIN {X 0,Y 545.059,Z 44.586,A -85,B 0,C 180,E1 -3816.995,E2 -3816.995} C_VEL
LIN {X 0,Y 544.353,Z 44.675,A -85,B 0,C 180,E1 -3817.611,E2 -3817.611} C_VEL
LIN {X 0,Y 541.493,Z 45.033,A -85,B 0,C 180,E1 -3818.612,E2 -3818.612} C_VEL
LIN {X 0,Y 539.104,Z 45.33,A -85,B 0,C 180,E1 -3819.418,E2 -3819.418} C_VEL
LIN {X 0,Y 538.086,Z 45.461,A -85,B 0,C 180,E1 -3820.04,E2 -3820.04} C_VEL
LIN {X 0,Y 538.006,Z 45.463,A -85,B 0,C 180,E1 -3820.251,E2 -3820.251} C_VEL
LIN {X 0,Y 538,Z 45.466,A -85,B 0,C 180,E1 -3822.984,E2 -3822.984} C_VEL
LIN {X 0,Y 538.013,Z 45.472,A -85,B 0,C 180,E1 -3825.927,E2 -3825.927} C_VEL
LIN {X 0,Y 538.05,Z 45.461,A -85,B 0,C 180,E1 -3829.253,E2 -3829.253} C_VEL
LIN {X 0,Y 537.987,Z 45.471,A -85,B 0,C 180,E1 -3832.122,E2 -3832.122} C_VEL
LIN {X 0,Y 537.995,Z 45.468,A -85,B 0,C 180,E1 -3834.915,E2 -3834.915} C_VEL
LIN {X 0,Y 538.017,Z 45.472,A -85,B 0,C 180,E1 -3837.617,E2 -3837.617} C_VEL
LIN {X 0,Y 538.008,Z 45.468,A -85,B 0,C 180,E1 -3840.238,E2 -3840.238} C_VEL
LIN {X 0,Y 538.088,Z 45.591,A -85,B 0,C 180,E1 -3841.873,E2 -3841.873} C_VEL
LIN {X 0,Y 538.426,Z 50.174,A -85,B 0,C 180,E1 -3842.816,E2 -3842.816} C_VEL
LIN {X 0,Y 538.257,Z 62.574,A -85,B 0,C 180,E1 -3845.303,E2 -3845.303} C_VEL
LIN {X 0,Y 539.742,Z 70.731,A -85,B 0,C 180,E1 -3845.468,E2 -3845.468} C_VEL
LIN {X 0,Y 539.333,Z 168.211,A -85,B 0,C 180,E1 -3846.785,E2 -3846.785} C_VEL
LIN {X 0,Y 539.212,Z 181.35,A -85,B 0,C 180,E1 -3847.109,E2 -3847.109} C_VEL
LIN {X 0,Y 539.087,Z 194.151,A -85,B 0,C 180,E1 -3847.584,E2 -3847.584} C_VEL
LIN {X 0,Y 538.825,Z 205.969,A -85,B 0,C 180,E1 -3848.177,E2 -3848.177} C_VEL
LIN {X 0,Y 538.586,Z 216.652,A -85,B 0,C 180,E1 -3848.87,E2 -3848.87} C_VEL
LIN {X 0,Y 538.423,Z 226.842,A -85,B 0,C 180,E1 -3849.693,E2 -3849.693} C_VEL
LIN {X 0,Y 538.192,Z 235.555,A -85,B 0,C 180,E1 -3850.549,E2 -3850.549} C_VEL
LIN {X 0,Y 537.994,Z 243.796,A -85,B 0,C 180,E1 -3851.531,E2 -3851.531} C_VEL
LIN {X 0,Y 537.865,Z 251.299,A -85,B 0,C 180,E1 -3852.627,E2 -3852.627} C_VEL
LIN {X 0,Y 537.736,Z 257.141,A -85,B 0,C 180,E1 -3853.68,E2 -3853.68} C_VEL
LIN {X 0,Y 537.664,Z 262.29,A -85,B 0,C 180,E1 -3854.845,E2 -3854.845} C_VEL
LIN {X 0,Y 537.606,Z 266.239,A -85,B 0,C 180,E1 -3856.004,E2 -3856.004} C_VEL
LIN {X 0,Y 537.53,Z 269.107,A -85,B 0,C 180,E1 -3857.158,E2 -3857.158} C_VEL
LIN {X 0,Y 537.521,Z 270.447,A -85,B 0,C 180,E1 -3857.925,E2 -3857.925} C_VEL
LIN {X 0,Y 537.539,Z 271.383,A -85,B 0,C 180,E1 -3858.69,E2 -3858.69} C_VEL
LIN {X 0,Y 537.503,Z 271.918,A -85,B 0,C 180,E1 -3859.452,E2 -3859.452} C_VEL
LIN {X 0,Y 537.512,Z 272.009,A -85,B 0,C 180,E1 -3860.214,E2 -3860.214} C_VEL
LIN {X 0,Y 537.543,Z 271.026,A -85,B 0,C 180,E1 -3861.731,E2 -3861.731} C_VEL
LIN {X 0,Y 537.55,Z 269.942,A -85,B 0,C 180,E1 -3862.488,E2 -3862.488} C_VEL
LIN {X 0,Y 537.606,Z 267.853,A -85,B 0,C 180,E1 -3863.479,E2 -3863.479} C_VEL
LIN {X 0,Y 537.595,Z 264.116,A -85,B 0,C 180,E1 -3864.749,E2 -3864.749} C_VEL
LIN {X 0,Y 537.725,Z 259.634,A -85,B 0,C 180,E1 -3865.878,E2 -3865.878} C_VEL
LIN {X 0,Y 537.768,Z 252.878,A -85,B 0,C 180,E1 -3867.191,E2 -3867.191} C_VEL
LIN {X 0,Y 537.944,Z 245.56,A -85,B 0,C 180,E1 -3868.316,E2 -3868.316} C_VEL
LIN {X 0,Y 538.164,Z 238.11,A -85,B 0,C 180,E1 -3869.252,E2 -3869.252} C_VEL
LIN {X 0,Y 538.29,Z 229.146,A -85,B 0,C 180,E1 -3870.187,E2 -3870.187} C_VEL
LIN {X 0,Y 538.519,Z 219.205,A -85,B 0,C 180,E1 -3871.028,E2 -3871.028} C_VEL
LIN {X 0,Y 538.787,Z 208.193,A -85,B 0,C 180,E1 -3871.775,E2 -3871.775} C_VEL
LIN {X 0,Y 539.027,Z 195.878,A -85,B 0,C 180,E1 -3872.429,E2 -3872.429} C_VEL
LIN {X 0,Y 539.192,Z 183.303,A -85,B 0,C 180,E1 -3872.919,E2 -3872.919} C_VEL
LIN {X 0,Y 539.321,Z 171.059,A -85,B 0,C 180,E1 -3873.245,E2 -3873.245} C_VEL
LIN {X 0,Y 539.45,Z 150.949,A -85,B 0,C 180,E1 -3873.548,E2 -3873.548} C_VEL
LIN {X 0,Y 539.6,Z 69.216,A -85,B 0,C 180,E1 -3874.646,E2 -3874.646} C_VEL
LIN {X 0,Y 538.232,Z 62.423,A -85,B 0,C 180,E1 -3874.799,E2 -3874.799} C_VEL
LIN {X 0,Y 538.481,Z 50.022,A -85,B 0,C 180,E1 -3877.29,E2 -3877.29} C_VEL
LIN {X 0,Y 538.084,Z 45.462,A -85,B 0,C 180,E1 -3878.261,E2 -3878.261} C_VEL
LIN {X 0,Y 538.092,Z 45.453,A -85,B 0,C 180,E1 -3881.601,E2 -3881.601} C_VEL
LIN {X 0,Y 538.061,Z 45.461,A -85,B 0,C 180,E1 -3884.857,E2 -3884.857} C_VEL
LIN {X 0,Y 538.062,Z 45.457,A -85,B 0,C 180,E1 -3887.541,E2 -3887.541} C_VEL
LIN {X 0,Y 538.04,Z 45.464,A -85,B 0,C 180,E1 -3890.652,E2 -3890.652} C_VEL
LIN {X 0,Y 538.005,Z 45.468,A -85,B 0,C 180,E1 -3893.889,E2 -3893.889} C_VEL
LIN {X 0,Y 538.044,Z 45.465,A -85,B 0,C 180,E1 -3896.367,E2 -3896.367} C_VEL
LIN {X 0,Y 538.033,Z 45.46,A -85,B 0,C 180,E1 -3898.934,E2 -3898.934} C_VEL
LIN {X 0,Y 538.013,Z 45.471,A -85,B 0,C 180,E1 -3901.887,E2 -3901.887} C_VEL
LIN {X 0,Y 538.03,Z 45.461,A -85,B 0,C 180,E1 -3904.62,E2 -3904.62} C_VEL
LIN {X 0,Y 538.009,Z 45.465,A -85,B 0,C 180,E1 -3907.17,E2 -3907.17} C_VEL
LIN {X 0,Y 538.026,Z 45.468,A -85,B 0,C 180,E1 -3909.797,E2 -3909.797} C_VEL
LIN {X 0,Y 538.021,Z 45.462,A -85,B 0,C 180,E1 -3912.786,E2 -3912.786} C_VEL
LIN {X 0,Y 538.021,Z 45.464,A -85,B 0,C 180,E1 -3915.927,E2 -3915.927} C_VEL
LIN {X 0,Y 538.034,Z 45.46,A -85,B 0,C 180,E1 -3918.227,E2 -3918.227} C_VEL
LIN {X 0,Y 538.017,Z 45.47,A -85,B 0,C 180,E1 -3921.17,E2 -3921.17} C_VEL
LIN {X 0,Y 537.998,Z 45.465,A -85,B 0,C 180,E1 -3924.089,E2 -3924.089} C_VEL
LIN {X 0,Y 538.034,Z 45.464,A -85,B 0,C 180,E1 -3926.728,E2 -3926.728} C_VEL
LIN {X 0,Y 538.031,Z 45.462,A -85,B 0,C 180,E1 -3929.557,E2 -3929.557} C_VEL
LIN {X 0,Y 538.045,Z 45.459,A -85,B 0,C 180,E1 -3931.95,E2 -3931.95} C_VEL
LIN {X 0,Y 538.075,Z 45.459,A -85,B 0,C 180,E1 -3934.467,E2 -3934.467} C_VEL
LIN {X 0,Y 537.999,Z 45.465,A -85,B 0,C 180,E1 -3937.739,E2 -3937.739} C_VEL
LIN {X 0,Y 538.085,Z 45.457,A -85,B 0,C 180,E1 -3940.148,E2 -3940.148} C_VEL
LIN {X 0,Y 538.017,Z 45.462,A -85,B 0,C 180,E1 -3943.299,E2 -3943.299} C_VEL
LIN {X 0,Y 538.069,Z 45.456,A -85,B 0,C 180,E1 -3945.631,E2 -3945.631} C_VEL
LIN {X 0,Y 538.084,Z 45.457,A -85,B 0,C 180,E1 -3948.702,E2 -3948.702} C_VEL
LIN {X 0,Y 538.066,Z 45.459,A -85,B 0,C 180,E1 -3951.739,E2 -3951.739} C_VEL
LIN {X 0,Y 538.127,Z 45.457,A -85,B 0,C 180,E1 -3954.003,E2 -3954.003} C_VEL
LIN {X 0,Y 538.14,Z 45.447,A -85,B 0,C 180,E1 -3957.006,E2 -3957.006} C_VEL
LIN {X 0,Y 538.178,Z 45.449,A -85,B 0,C 180,E1 -3960,E2 -3960} C_VEL
LIN {X 0,Y 538.14,Z 45.447,A -85,B 0,C 180,E1 -3962.995,E2 -3962.995} C_VEL
LIN {X 0,Y 538.097,Z 45.456,A -85,B 0,C 180,E1 -3965.998,E2 -3965.998} C_VEL
LIN {X 0,Y 538.059,Z 45.459,A -85,B 0,C 180,E1 -3969.018,E2 -3969.018} C_VEL
LIN {X 0,Y 538.072,Z 45.456,A -85,B 0,C 180,E1 -3972.063,E2 -3972.063} C_VEL
LIN {X 0,Y 538.051,Z 45.465,A -85,B 0,C 180,E1 -3975.144,E2 -3975.144} C_VEL
LIN {X 0,Y 538.022,Z 45.462,A -85,B 0,C 180,E1 -3978.271,E2 -3978.271} C_VEL
LIN {X 0,Y 538.043,Z 45.462,A -85,B 0,C 180,E1 -3980.651,E2 -3980.651} C_VEL
LIN {X 0,Y 538.007,Z 45.464,A -85,B 0,C 180,E1 -3983.888,E2 -3983.888} C_VEL
LIN {X 0,Y 538.042,Z 45.461,A -85,B 0,C 180,E1 -3986.367,E2 -3986.367} C_VEL
LIN {X 0,Y 538.035,Z 45.467,A -85,B 0,C 180,E1 -3988.933,E2 -3988.933} C_VEL
LIN {X 0,Y 538.015,Z 45.463,A -85,B 0,C 180,E1 -3991.887,E2 -3991.887} C_VEL
LIN {X 0,Y 538.013,Z 45.472,A -85,B 0,C 180,E1 -3994.617,E2 -3994.617} C_VEL
LIN {X 0,Y 538.004,Z 45.465,A -85,B 0,C 180,E1 -3997.169,E2 -3997.169} C_VEL
LIN {X 0,Y 538.026,Z 45.462,A -85,B 0,C 180,E1 -3999.797,E2 -3999.797} C_VEL
LIN {X 0,Y 538.023,Z 45.464,A -85,B 0,C 180,E1 -4002.786,E2 -4002.786} C_VEL
LIN {X 0,Y 538.015,Z 45.468,A -85,B 0,C 180,E1 -4005.927,E2 -4005.927} C_VEL
LIN {X 0,Y 538.052,Z 45.458,A -85,B 0,C 180,E1 -4009.253,E2 -4009.253} C_VEL
LIN {X 0,Y 537.993,Z 45.472,A -85,B 0,C 180,E1 -4012.122,E2 -4012.122} C_VEL
LIN {X 0,Y 537.998,Z 45.465,A -85,B 0,C 180,E1 -4014.915,E2 -4014.915} C_VEL
LIN {X 0,Y 538.02,Z 45.469,A -85,B 0,C 180,E1 -4017.617,E2 -4017.617} C_VEL
LIN {X 0,Y 538.018,Z 45.466,A -85,B 0,C 180,E1 -4020.239,E2 -4020.239} C_VEL
LIN {X 0,Y 538.057,Z 45.46,A -85,B 0,C 180,E1 -4022.795,E2 -4022.795} C_VEL
LIN {X 0,Y 538.09,Z 45.553,A -85,B 0,C 180,E1 -4025.037,E2 -4025.037} C_VEL
LIN {X 0,Y 539.328,Z 52.967,A -85,B 0,C 180,E1 -4026.174,E2 -4026.174} C_VEL
LIN {X 0,Y 538.995,Z 71.063,A -85,B 0,C 180,E1 -4028.787,E2 -4028.787} C_VEL
LIN {X 0,Y 538.663,Z 91.896,A -85,B 0,C 180,E1 -4031.752,E2 -4031.752} C_VEL
LIN {X 0,Y 538.319,Z 112.676,A -85,B 0,C 180,E1 -4034.67,E2 -4034.67} C_VEL
LIN {X 0,Y 538.243,Z 116.752,A -85,B 0,C 180,E1 -4035.238,E2 -4035.238} C_VEL
LIN {X 0,Y 539.64,Z 126.981,A -85,B 0,C 180,E1 -4035.415,E2 -4035.415} C_VEL
LIN {X 0,Y 539.282,Z 225.426,A -85,B 0,C 180,E1 -4036.745,E2 -4036.745} C_VEL
LIN {X 0,Y 539.073,Z 238.759,A -85,B 0,C 180,E1 -4037.075,E2 -4037.075} C_VEL
LIN {X 0,Y 538.922,Z 250.972,A -85,B 0,C 180,E1 -4037.526,E2 -4037.526} C_VEL
LIN {X 0,Y 538.66,Z 262.749,A -85,B 0,C 180,E1 -4038.109,E2 -4038.109} C_VEL
LIN {X 0,Y 538.424,Z 274.938,A -85,B 0,C 180,E1 -4038.899,E2 -4038.899} C_VEL
LIN {X 0,Y 538.189,Z 285.425,A -85,B 0,C 180,E1 -4039.751,E2 -4039.751} C_VEL
LIN {X 0,Y 538.023,Z 294.004,A -85,B 0,C 180,E1 -4040.602,E2 -4040.602} C_VEL
LIN {X 0,Y 537.876,Z 301.923,A -85,B 0,C 180,E1 -4041.547,E2 -4041.547} C_VEL
LIN {X 0,Y 537.711,Z 309.657,A -85,B 0,C 180,E1 -4042.679,E2 -4042.679} C_VEL
LIN {X 0,Y 537.644,Z 316.792,A -85,B 0,C 180,E1 -4043.997,E2 -4043.997} C_VEL
LIN {X 0,Y 537.539,Z 321.535,A -85,B 0,C 180,E1 -4045.125,E2 -4045.125} C_VEL
LIN {X 0,Y 537.591,Z 325.167,A -85,B 0,C 180,E1 -4046.252,E2 -4046.252} C_VEL
LIN {X 0,Y 537.58,Z 327.038,A -85,B 0,C 180,E1 -4047.002,E2 -4047.002} C_VEL
LIN {X 0,Y 537.461,Z 329.436,A -85,B 0,C 180,E1 -4048.501,E2 -4048.501} C_VEL
LIN {X 0,Y 537.46,Z 330.046,A -85,B 0,C 180,E1 -4049.251,E2 -4049.251} C_VEL
LIN {X 0,Y 537.461,Z 330.263,A -85,B 0,C 180,E1 -4050,E2 -4050} C_VEL
LIN {X 0,Y 537.46,Z 330.045,A -85,B 0,C 180,E1 -4050.749,E2 -4050.749} C_VEL
LIN {X 0,Y 537.49,Z 328.434,A -85,B 0,C 180,E1 -4052.248,E2 -4052.248} C_VEL
LIN {X 0,Y 537.58,Z 327.035,A -85,B 0,C 180,E1 -4052.998,E2 -4052.998} C_VEL
LIN {X 0,Y 537.603,Z 324.083,A -85,B 0,C 180,E1 -4054.123,E2 -4054.123} C_VEL
LIN {X 0,Y 537.587,Z 320.084,A -85,B 0,C 180,E1 -4055.251,E2 -4055.251} C_VEL
LIN {X 0,Y 537.64,Z 314.031,A -85,B 0,C 180,E1 -4056.551,E2 -4056.551} C_VEL
LIN {X 0,Y 537.749,Z 307.227,A -85,B 0,C 180,E1 -4057.698,E2 -4057.698} C_VEL
LIN {X 0,Y 537.909,Z 298.902,A -85,B 0,C 180,E1 -4058.831,E2 -4058.831} C_VEL
LIN {X 0,Y 538.057,Z 290.371,A -85,B 0,C 180,E1 -4059.776,E2 -4059.776} C_VEL
LIN {X 0,Y 538.293,Z 279.837,A -85,B 0,C 180,E1 -4060.722,E2 -4060.722} C_VEL
LIN {X 0,Y 538.521,Z 268.74,A -85,B 0,C 180,E1 -4061.525,E2 -4061.525} C_VEL
LIN {X 0,Y 538.779,Z 258.008,A -85,B 0,C 180,E1 -4062.142,E2 -4062.142} C_VEL
LIN {X 0,Y 539.004,Z 246.299,A -85,B 0,C 180,E1 -4062.663,E2 -4062.663} C_VEL
LIN {X 0,Y 539.169,Z 232.812,A -85,B 0,C 180,E1 -4063.09,E2 -4063.09} C_VEL
LIN {X 0,Y 539.354,Z 219.47,A -85,B 0,C 180,E1 -4063.349,E2 -4063.349} C_VEL
LIN {X 0,Y 539.465,Z 125.367,A -85,B 0,C 180,E1 -4064.61,E2 -4064.61} C_VEL
LIN {X 0,Y 538.228,Z 116.568,A -85,B 0,C 180,E1 -4064.779,E2 -4064.779} C_VEL
LIN {X 0,Y 538.578,Z 95.596,A -85,B 0,C 180,E1 -4067.713,E2 -4067.713} C_VEL
LIN {X 0,Y 538.913,Z 75.111,A -85,B 0,C 180,E1 -4070.616,E2 -4070.616} C_VEL
LIN {X 0,Y 539.371,Z 52.861,A -85,B 0,C 180,E1 -4073.824,E2 -4073.824} C_VEL
LIN {X 0,Y 538.087,Z 45.46,A -85,B 0,C 180,E1 -4074.989,E2 -4074.989} C_VEL
LIN {X 0,Y 538.043,Z 45.467,A -85,B 0,C 180,E1 -4078.05,E2 -4078.05} C_VEL
LIN {X 0,Y 538.024,Z 45.466,A -85,B 0,C 180,E1 -4080.627,E2 -4080.627} C_VEL
LIN {X 0,Y 538.022,Z 45.463,A -85,B 0,C 180,E1 -4083.278,E2 -4083.278} C_VEL
LIN {X 0,Y 537.998,Z 45.474,A -85,B 0,C 180,E1 -4086.005,E2 -4086.005} C_VEL
LIN {X 0,Y 538.016,Z 45.461,A -85,B 0,C 180,E1 -4088.831,E2 -4088.831} C_VEL
LIN {X 0,Y 538.034,Z 45.469,A -85,B 0,C 180,E1 -4091.773,E2 -4091.773} C_VEL
LIN {X 0,Y 538.008,Z 45.463,A -85,B 0,C 180,E1 -4094.862,E2 -4094.862} C_VEL
LIN {X 0,Y 538.022,Z 45.465,A -85,B 0,C 180,E1 -4097.214,E2 -4097.214} C_VEL
LIN {X 0,Y 538.026,Z 45.46,A -85,B 0,C 180,E1 -4100.203,E2 -4100.203} C_VEL
LIN {X 0,Y 538.028,Z 45.465,A -85,B 0,C 180,E1 -4103.067,E2 -4103.067} C_VEL
LIN {X 0,Y 538.015,Z 45.463,A -85,B 0,C 180,E1 -4105.826,E2 -4105.826} C_VEL
LIN {X 0,Y 538.013,Z 45.465,A -85,B 0,C 180,E1 -4108.499,E2 -4108.499} C_VEL
LIN {X 0,Y 538.065,Z 45.465,A -85,B 0,C 180,E1 -4111.1,E2 -4111.1} C_VEL
LIN {X 0,Y 538.046,Z 45.458,A -85,B 0,C 180,E1 -4113.633,E2 -4113.633} C_VEL
LIN {X 0,Y 538.011,Z 45.464,A -85,B 0,C 180,E1 -4116.122,E2 -4116.122} C_VEL
LIN {X 0,Y 538.042,Z 45.46,A -85,B 0,C 180,E1 -4119.349,E2 -4119.349} C_VEL
LIN {X 0,Y 538.06,Z 45.464,A -85,B 0,C 180,E1 -4122.517,E2 -4122.517} C_VEL
LIN {X 0,Y 538.069,Z 45.457,A -85,B 0,C 180,E1 -4125.631,E2 -4125.631} C_VEL
LIN {X 0,Y 538.083,Z 45.457,A -85,B 0,C 180,E1 -4128.702,E2 -4128.702} C_VEL
LIN {X 0,Y 538.088,Z 45.457,A -85,B 0,C 180,E1 -4131.74,E2 -4131.74} C_VEL
LIN {X 0,Y 538.163,Z 45.445,A -85,B 0,C 180,E1 -4134.755,E2 -4134.755} C_VEL
LIN {X 0,Y 538.17,Z 45.45,A -85,B 0,C 180,E1 -4137.755,E2 -4137.755} C_VEL
LIN {X 0,Y 538.185,Z 45.442,A -85,B 0,C 180,E1 -4140.748,E2 -4140.748} C_VEL
LIN {X 0,Y 538.139,Z 45.447,A -85,B 0,C 180,E1 -4142.994,E2 -4142.994} C_VEL
LIN {X 0,Y 538.095,Z 45.456,A -85,B 0,C 180,E1 -4145.998,E2 -4145.998} C_VEL
LIN {X 0,Y 538.057,Z 45.458,A -85,B 0,C 180,E1 -4149.018,E2 -4149.018} C_VEL
LIN {X 0,Y 538.088,Z 45.454,A -85,B 0,C 180,E1 -4152.062,E2 -4152.062} C_VEL
LIN {X 0,Y 538.05,Z 45.465,A -85,B 0,C 180,E1 -4155.144,E2 -4155.144} C_VEL
LIN {X 0,Y 538.02,Z 45.461,A -85,B 0,C 180,E1 -4158.271,E2 -4158.271} C_VEL
LIN {X 0,Y 538.042,Z 45.463,A -85,B 0,C 180,E1 -4160.651,E2 -4160.651} C_VEL
LIN {X 0,Y 538.005,Z 45.463,A -85,B 0,C 180,E1 -4163.888,E2 -4163.888} C_VEL
LIN {X 0,Y 538.039,Z 45.463,A -85,B 0,C 180,E1 -4166.367,E2 -4166.367} C_VEL
LIN {X 0,Y 538.033,Z 45.465,A -85,B 0,C 180,E1 -4168.933,E2 -4168.933} C_VEL
LIN {X 0,Y 538.013,Z 45.464,A -85,B 0,C 180,E1 -4171.887,E2 -4171.887} C_VEL
LIN {X 0,Y 538.009,Z 45.47,A -85,B 0,C 180,E1 -4174.616,E2 -4174.616} C_VEL
LIN {X 0,Y 538.001,Z 45.464,A -85,B 0,C 180,E1 -4177.169,E2 -4177.169} C_VEL
LIN {X 0,Y 538.023,Z 45.465,A -85,B 0,C 180,E1 -4179.797,E2 -4179.797} C_VEL
LIN {X 0,Y 538.006,Z 45.463,A -85,B 0,C 180,E1 -4180.251,E2 -4180.251} C_VEL
LIN {X 0,Y 537.345,Z 45.545,A -85,B 0,C 180,E1 -4180.876,E2 -4180.876} C_VEL
LIN {X 0,Y 534.492,Z 45.904,A -85,B 0,C 180,E1 -4181.891,E2 -4181.891} C_VEL
LIN {X 0,Y 532.074,Z 46.208,A -85,B 0,C 180,E1 -4182.708,E2 -4182.708} C_VEL
LIN {X 0,Y 531.031,Z 46.336,A -85,B 0,C 180,E1 -4183.339,E2 -4183.339} C_VEL
LIN {X 0,Y 530.945,Z 46.346,A -85,B 0,C 180,E1 -4183.553,E2 -4183.553} C_VEL
LIN {X 0,Y 530.939,Z 46.347,A -85,B 0,C 180,E1 -4186.502,E2 -4186.502} C_VEL
LIN {X 0,Y 530.984,Z 46.34,A -85,B 0,C 180,E1 -4188.977,E2 -4188.977} C_VEL
LIN {X 0,Y 530.953,Z 46.349,A -85,B 0,C 180,E1 -4191.529,E2 -4191.529} C_VEL
LIN {X 0,Y 530.951,Z 46.345,A -85,B 0,C 180,E1 -4194.379,E2 -4194.379} C_VEL
LIN {X 0,Y 530.968,Z 46.348,A -85,B 0,C 180,E1 -4197.133,E2 -4197.133} C_VEL
LIN {X 0,Y 530.954,Z 46.35,A -85,B 0,C 180,E1 -4199.802,E2 -4199.802} C_VEL
LIN {X 0,Y 531.085,Z 46.526,A -85,B 0,C 180,E1 -4201.765,E2 -4201.765} C_VEL
LIN {X 0,Y 531.426,Z 51.782,A -85,B 0,C 180,E1 -4202.854,E2 -4202.854} C_VEL
LIN {X 0,Y 531.284,Z 62.879,A -85,B 0,C 180,E1 -4205.099,E2 -4205.099} C_VEL
LIN {X 0,Y 532.856,Z 70.411,A -85,B 0,C 180,E1 -4205.265,E2 -4205.265} C_VEL
LIN {X 0,Y 532.444,Z 169.118,A -85,B 0,C 180,E1 -4206.621,E2 -4206.621} C_VEL
LIN {X 0,Y 532.312,Z 182.867,A -85,B 0,C 180,E1 -4206.975,E2 -4206.975} C_VEL
LIN {X 0,Y 532.173,Z 194.78,A -85,B 0,C 180,E1 -4207.43,E2 -4207.43} C_VEL
LIN {X 0,Y 531.884,Z 206.438,A -85,B 0,C 180,E1 -4208.026,E2 -4208.026} C_VEL
LIN {X 0,Y 531.602,Z 217.843,A -85,B 0,C 180,E1 -4208.782,E2 -4208.782} C_VEL
LIN {X 0,Y 531.403,Z 228.669,A -85,B 0,C 180,E1 -4209.686,E2 -4209.686} C_VEL
LIN {X 0,Y 531.155,Z 238.259,A -85,B 0,C 180,E1 -4210.683,E2 -4210.683} C_VEL
LIN {X 0,Y 530.906,Z 247.453,A -85,B 0,C 180,E1 -4211.875,E2 -4211.875} C_VEL
LIN {X 0,Y 530.763,Z 254.764,A -85,B 0,C 180,E1 -4213.064,E2 -4213.064} C_VEL
LIN {X 0,Y 530.658,Z 260.511,A -85,B 0,C 180,E1 -4214.246,E2 -4214.246} C_VEL
LIN {X 0,Y 530.574,Z 264.983,A -85,B 0,C 180,E1 -4215.423,E2 -4215.423} C_VEL
LIN {X 0,Y 530.512,Z 267.328,A -85,B 0,C 180,E1 -4216.205,E2 -4216.205} C_VEL
LIN {X 0,Y 530.464,Z 269.225,A -85,B 0,C 180,E1 -4216.984,E2 -4216.984} C_VEL
LIN {X 0,Y 530.451,Z 270.635,A -85,B 0,C 180,E1 -4217.761,E2 -4217.761} C_VEL
LIN {X 0,Y 530.448,Z 271.744,A -85,B 0,C 180,E1 -4218.649,E2 -4218.649} C_VEL
LIN {X 0,Y 530.43,Z 272.42,A -85,B 0,C 180,E1 -4220.082,E2 -4220.082} C_VEL
LIN {X 0,Y 530.451,Z 271.55,A -85,B 0,C 180,E1 -4221.62,E2 -4221.62} C_VEL
LIN {X 0,Y 530.474,Z 270.535,A -85,B 0,C 180,E1 -4222.387,E2 -4222.387} C_VEL
LIN {X 0,Y 530.548,Z 268.374,A -85,B 0,C 180,E1 -4223.464,E2 -4223.464} C_VEL
LIN {X 0,Y 530.524,Z 264.925,A -85,B 0,C 180,E1 -4224.679,E2 -4224.679} C_VEL
LIN {X 0,Y 530.655,Z 260.573,A -85,B 0,C 180,E1 -4225.823,E2 -4225.823} C_VEL
LIN {X 0,Y 530.695,Z 255.068,A -85,B 0,C 180,E1 -4226.964,E2 -4226.964} C_VEL
LIN {X 0,Y 530.885,Z 248.194,A -85,B 0,C 180,E1 -4228.103,E2 -4228.103} C_VEL
LIN {X 0,Y 531.136,Z 239.602,A -85,B 0,C 180,E1 -4229.242,E2 -4229.242} C_VEL
LIN {X 0,Y 531.29,Z 230.853,A -85,B 0,C 180,E1 -4230.19,E2 -4230.19} C_VEL
LIN {X 0,Y 531.561,Z 220.071,A -85,B 0,C 180,E1 -4231.136,E2 -4231.136} C_VEL
LIN {X 0,Y 531.844,Z 209.172,A -85,B 0,C 180,E1 -4231.893,E2 -4231.893} C_VEL
LIN {X 0,Y 532.096,Z 197.011,A -85,B 0,C 180,E1 -4232.555,E2 -4232.555} C_VEL
LIN {X 0,Y 532.255,Z 185.505,A -85,B 0,C 180,E1 -4233.028,E2 -4233.028} C_VEL
LIN {X 0,Y 532.404,Z 173.18,A -85,B 0,C 180,E1 -4233.382,E2 -4233.382} C_VEL
LIN {X 0,Y 532.512,Z 157.585,A -85,B 0,C 180,E1 -4233.642,E2 -4233.642} C_VEL
LIN {X 0,Y 532.822,Z 70.478,A -85,B 0,C 180,E1 -4234.824,E2 -4234.824} C_VEL
LIN {X 0,Y 531.25,Z 62.835,A -85,B 0,C 180,E1 -4234.981,E2 -4234.981} C_VEL
LIN {X 0,Y 531.509,Z 50.943,A -85,B 0,C 180,E1 -4237.385,E2 -4237.385} C_VEL
LIN {X 0,Y 531.054,Z 46.338,A -85,B 0,C 180,E1 -4238.371,E2 -4238.371} C_VEL
LIN {X 0,Y 531.054,Z 46.329,A -85,B 0,C 180,E1 -4241.672,E2 -4241.672} C_VEL
LIN {X 0,Y 531.033,Z 46.336,A -85,B 0,C 180,E1 -4244.956,E2 -4244.956} C_VEL
LIN {X 0,Y 531.019,Z 46.335,A -85,B 0,C 180,E1 -4247.722,E2 -4247.722} C_VEL
LIN {X 0,Y 531.027,Z 46.338,A -85,B 0,C 180,E1 -4250.127,E2 -4250.127} C_VEL
LIN {X 0,Y 530.947,Z 46.348,A -85,B 0,C 180,E1 -4252.574,E2 -4252.574} C_VEL
LIN {X 0,Y 530.997,Z 46.337,A -85,B 0,C 180,E1 -4255.058,E2 -4255.058} C_VEL
LIN {X 0,Y 531.018,Z 46.336,A -85,B 0,C 180,E1 -4257.596,E2 -4257.596} C_VEL
LIN {X 0,Y 530.977,Z 46.34,A -85,B 0,C 180,E1 -4260.645,E2 -4260.645} C_VEL
LIN {X 0,Y 530.992,Z 46.345,A -85,B 0,C 180,E1 -4263.773,E2 -4263.773} C_VEL
LIN {X 0,Y 530.968,Z 46.341,A -85,B 0,C 180,E1 -4266.558,E2 -4266.558} C_VEL
LIN {X 0,Y 530.981,Z 46.345,A -85,B 0,C 180,E1 -4269.854,E2 -4269.854} C_VEL
LIN {X 0,Y 530.981,Z 46.339,A -85,B 0,C 180,E1 -4272.457,E2 -4272.457} C_VEL
LIN {X 0,Y 530.979,Z 46.345,A -85,B 0,C 180,E1 -4275.622,E2 -4275.622} C_VEL
LIN {X 0,Y 530.996,Z 46.337,A -85,B 0,C 180,E1 -4278.565,E2 -4278.565} C_VEL
LIN {X 0,Y 530.961,Z 46.346,A -85,B 0,C 180,E1 -4281.53,E2 -4281.53} C_VEL
LIN {X 0,Y 530.959,Z 46.342,A -85,B 0,C 180,E1 -4284.38,E2 -4284.38} C_VEL
LIN {X 0,Y 530.971,Z 46.348,A -85,B 0,C 180,E1 -4287.134,E2 -4287.134} C_VEL
LIN {X 0,Y 530.974,Z 46.34,A -85,B 0,C 180,E1 -4289.803,E2 -4289.803} C_VEL
LIN {X 0,Y 531.017,Z 46.338,A -85,B 0,C 180,E1 -4292.468,E2 -4292.468} C_VEL
LIN {X 0,Y 531,Z 46.343,A -85,B 0,C 180,E1 -4294.942,E2 -4294.942} C_VEL
LIN {X 0,Y 530.977,Z 46.343,A -85,B 0,C 180,E1 -4298.247,E2 -4298.247} C_VEL
LIN {X 0,Y 530.99,Z 46.345,A -85,B 0,C 180,E1 -4300.677,E2 -4300.677} C_VEL
LIN {X 0,Y 530.975,Z 46.341,A -85,B 0,C 180,E1 -4303.071,E2 -4303.071} C_VEL
LIN {X 0,Y 531.025,Z 46.333,A -85,B 0,C 180,E1 -4305.436,E2 -4305.436} C_VEL
LIN {X 0,Y 531.043,Z 46.336,A -85,B 0,C 180,E1 -4308.55,E2 -4308.55} C_VEL
LIN {X 0,Y 531.041,Z 46.333,A -85,B 0,C 180,E1 -4311.629,E2 -4311.629} C_VEL
LIN {X 0,Y 531.123,Z 46.322,A -85,B 0,C 180,E1 -4314.685,E2 -4314.685} C_VEL
LIN {X 0,Y 531.143,Z 46.324,A -85,B 0,C 180,E1 -4317.725,E2 -4317.725} C_VEL
LIN {X 0,Y 531.157,Z 46.317,A -85,B 0,C 180,E1 -4320.758,E2 -4320.758} C_VEL
LIN {X 0,Y 531.107,Z 46.324,A -85,B 0,C 180,E1 -4323.034,E2 -4323.034} C_VEL
LIN {X 0,Y 531.056,Z 46.332,A -85,B 0,C 180,E1 -4326.078,E2 -4326.078} C_VEL
LIN {X 0,Y 531.021,Z 46.337,A -85,B 0,C 180,E1 -4329.138,E2 -4329.138} C_VEL
LIN {X 0,Y 531.056,Z 46.335,A -85,B 0,C 180,E1 -4331.671,E2 -4331.671} C_VEL
LIN {X 0,Y 531.037,Z 46.336,A -85,B 0,C 180,E1 -4334.956,E2 -4334.956} C_VEL
LIN {X 0,Y 530.986,Z 46.34,A -85,B 0,C 180,E1 -4337.724,E2 -4337.724} C_VEL
LIN {X 0,Y 531.031,Z 46.333,A -85,B 0,C 180,E1 -4340.127,E2 -4340.127} C_VEL
LIN {X 0,Y 530.95,Z 46.345,A -85,B 0,C 180,E1 -4342.573,E2 -4342.573} C_VEL
LIN {X 0,Y 530.994,Z 46.345,A -85,B 0,C 180,E1 -4345.058,E2 -4345.058} C_VEL
LIN {X 0,Y 530.978,Z 46.34,A -85,B 0,C 180,E1 -4347.598,E2 -4347.598} C_VEL
LIN {X 0,Y 530.975,Z 46.341,A -85,B 0,C 180,E1 -4350.197,E2 -4350.197} C_VEL
LIN {X 0,Y 530.971,Z 46.346,A -85,B 0,C 180,E1 -4352.867,E2 -4352.867} C_VEL
LIN {X 0,Y 530.955,Z 46.342,A -85,B 0,C 180,E1 -4355.62,E2 -4355.62} C_VEL
LIN {X 0,Y 530.969,Z 46.346,A -85,B 0,C 180,E1 -4358.653,E2 -4358.653} C_VEL
LIN {X 0,Y 530.998,Z 46.337,A -85,B 0,C 180,E1 -4361.435,E2 -4361.435} C_VEL
LIN {X 0,Y 530.975,Z 46.344,A -85,B 0,C 180,E1 -4364.548,E2 -4364.548} C_VEL
LIN {X 0,Y 530.974,Z 46.344,A -85,B 0,C 180,E1 -4367.836,E2 -4367.836} C_VEL
LIN {X 0,Y 530.975,Z 46.342,A -85,B 0,C 180,E1 -4370.555,E2 -4370.555} C_VEL
LIN {X 0,Y 530.954,Z 46.344,A -85,B 0,C 180,E1 -4373.441,E2 -4373.441} C_VEL
LIN {X 0,Y 530.961,Z 46.345,A -85,B 0,C 180,E1 -4376.225,E2 -4376.225} C_VEL
LIN {X 0,Y 530.97,Z 46.344,A -85,B 0,C 180,E1 -4379.356,E2 -4379.356} C_VEL
LIN {X 0,Y 531.015,Z 46.337,A -85,B 0,C 180,E1 -4382.468,E2 -4382.468} C_VEL
LIN {X 0,Y 531.078,Z 46.531,A -85,B 0,C 180,E1 -4384.894,E2 -4384.894} C_VEL
LIN {X 0,Y 532.373,Z 53.967,A -85,B 0,C 180,E1 -4386.05,E2 -4386.05} C_VEL
LIN {X 0,Y 531.999,Z 73.475,A -85,B 0,C 180,E1 -4388.9,E2 -4388.9} C_VEL
LIN {X 0,Y 531.637,Z 94.23,A -85,B 0,C 180,E1 -4391.891,E2 -4391.891} C_VEL
LIN {X 0,Y 531.287,Z 113.673,A -85,B 0,C 180,E1 -4394.659,E2 -4394.659} C_VEL
LIN {X 0,Y 531.206,Z 116.339,A -85,B 0,C 180,E1 -4395.035,E2 -4395.035} C_VEL
LIN {X 0,Y 532.779,Z 128.219,A -85,B 0,C 180,E1 -4395.245,E2 -4395.245} C_VEL
LIN {X 0,Y 532.387,Z 225.025,A -85,B 0,C 180,E1 -4396.57,E2 -4396.57} C_VEL
LIN {X 0,Y 532.151,Z 238.364,A -85,B 0,C 180,E1 -4396.904,E2 -4396.904} C_VEL
LIN {X 0,Y 531.952,Z 250.579,A -85,B 0,C 180,E1 -4397.36,E2 -4397.36} C_VEL
LIN {X 0,Y 531.662,Z 262.633,A -85,B 0,C 180,E1 -4397.967,E2 -4397.967} C_VEL
LIN {X 0,Y 531.43,Z 274.551,A -85,B 0,C 180,E1 -4398.751,E2 -4398.751} C_VEL
LIN {X 0,Y 531.191,Z 285.039,A -85,B 0,C 180,E1 -4399.615,E2 -4399.615} C_VEL
LIN {X 0,Y 530.958,Z 293.616,A -85,B 0,C 180,E1 -4400.476,E2 -4400.476} C_VEL
LIN {X 0,Y 530.784,Z 301.535,A -85,B 0,C 180,E1 -4401.433,E2 -4401.433} C_VEL
LIN {X 0,Y 530.642,Z 309.273,A -85,B 0,C 180,E1 -4402.58,E2 -4402.58} C_VEL
LIN {X 0,Y 530.537,Z 316.406,A -85,B 0,C 180,E1 -4403.917,E2 -4403.917} C_VEL
LIN {X 0,Y 530.458,Z 321.152,A -85,B 0,C 180,E1 -4405.06,E2 -4405.06} C_VEL
LIN {X 0,Y 530.516,Z 324.784,A -85,B 0,C 180,E1 -4406.202,E2 -4406.202} C_VEL
LIN {X 0,Y 530.512,Z 326.656,A -85,B 0,C 180,E1 -4406.962,E2 -4406.962} C_VEL
LIN {X 0,Y 530.37,Z 329.052,A -85,B 0,C 180,E1 -4408.481,E2 -4408.481} C_VEL
LIN {X 0,Y 530.37,Z 329.663,A -85,B 0,C 180,E1 -4409.241,E2 -4409.241} C_VEL
LIN {X 0,Y 530.372,Z 329.879,A -85,B 0,C 180,E1 -4410,E2 -4410} C_VEL
LIN {X 0,Y 530.37,Z 329.661,A -85,B 0,C 180,E1 -4410.759,E2 -4410.759} C_VEL
LIN {X 0,Y 530.412,Z 328.049,A -85,B 0,C 180,E1 -4412.278,E2 -4412.278} C_VEL
LIN {X 0,Y 530.512,Z 326.649,A -85,B 0,C 180,E1 -4413.038,E2 -4413.038} C_VEL
LIN {X 0,Y 530.521,Z 323.695,A -85,B 0,C 180,E1 -4414.178,E2 -4414.178} C_VEL
LIN {X 0,Y 530.52,Z 319.695,A -85,B 0,C 180,E1 -4415.321,E2 -4415.321} C_VEL
LIN {X 0,Y 530.538,Z 314.246,A -85,B 0,C 180,E1 -4416.525,E2 -4416.525} C_VEL
LIN {X 0,Y 530.66,Z 308.077,A -85,B 0,C 180,E1 -4417.611,E2 -4417.611} C_VEL
LIN {X 0,Y 530.811,Z 300.005,A -85,B 0,C 180,E1 -4418.758,E2 -4418.758} C_VEL
LIN {X 0,Y 530.97,Z 291.783,A -85,B 0,C 180,E1 -4419.716,E2 -4419.716} C_VEL
LIN {X 0,Y 531.262,Z 281.766,A -85,B 0,C 180,E1 -4420.673,E2 -4420.673} C_VEL
LIN {X 0,Y 531.463,Z 270.376,A -85,B 0,C 180,E1 -4421.543,E2 -4421.543} C_VEL
LIN {X 0,Y 531.779,Z 259.381,A -85,B 0,C 180,E1 -4422.208,E2 -4422.208} C_VEL
LIN {X 0,Y 532.015,Z 247.113,A -85,B 0,C 180,E1 -4422.784,E2 -4422.784} C_VEL
LIN {X 0,Y 532.234,Z 234.234,A -85,B 0,C 180,E1 -4423.215,E2 -4423.215} C_VEL
LIN {X 0,Y 532.438,Z 220.577,A -85,B 0,C 180,E1 -4423.501,E2 -4423.501} C_VEL
LIN {X 0,Y 532.616,Z 126.221,A -85,B 0,C 180,E1 -4424.785,E2 -4424.785} C_VEL
LIN {X 0,Y 531.208,Z 116.257,A -85,B 0,C 180,E1 -4424.966,E2 -4424.966} C_VEL
LIN {X 0,Y 531.597,Z 95.961,A -85,B 0,C 180,E1 -4427.846,E2 -4427.846} C_VEL
LIN {X 0,Y 531.987,Z 73.361,A -85,B 0,C 180,E1 -4431.1,E2 -4431.1} C_VEL
LIN {X 0,Y 532.402,Z 53.944,A -85,B 0,C 180,E1 -4433.949,E2 -4433.949} C_VEL
LIN {X 0,Y 531.032,Z 46.338,A -85,B 0,C 180,E1 -4435.161,E2 -4435.161} C_VEL
LIN {X 0,Y 531.016,Z 46.338,A -85,B 0,C 180,E1 -4437.596,E2 -4437.596} C_VEL
LIN {X 0,Y 530.977,Z 46.343,A -85,B 0,C 180,E1 -4440.645,E2 -4440.645} C_VEL
LIN {X 0,Y 530.961,Z 46.347,A -85,B 0,C 180,E1 -4443.775,E2 -4443.775} C_VEL
LIN {X 0,Y 530.958,Z 46.344,A -85,B 0,C 180,E1 -4446.559,E2 -4446.559} C_VEL
LIN {X 0,Y 530.989,Z 46.339,A -85,B 0,C 180,E1 -4449.443,E2 -4449.443} C_VEL
LIN {X 0,Y 530.981,Z 46.339,A -85,B 0,C 180,E1 -4452.457,E2 -4452.457} C_VEL
LIN {X 0,Y 530.979,Z 46.346,A -85,B 0,C 180,E1 -4455.622,E2 -4455.622} C_VEL
LIN {X 0,Y 530.997,Z 46.336,A -85,B 0,C 180,E1 -4458.564,E2 -4458.564} C_VEL
LIN {X 0,Y 530.961,Z 46.347,A -85,B 0,C 180,E1 -4461.529,E2 -4461.529} C_VEL
LIN {X 0,Y 530.958,Z 46.341,A -85,B 0,C 180,E1 -4464.38,E2 -4464.38} C_VEL
LIN {X 0,Y 530.97,Z 46.347,A -85,B 0,C 180,E1 -4467.133,E2 -4467.133} C_VEL
LIN {X 0,Y 530.974,Z 46.339,A -85,B 0,C 180,E1 -4469.803,E2 -4469.803} C_VEL
LIN {X 0,Y 531.017,Z 46.337,A -85,B 0,C 180,E1 -4472.468,E2 -4472.468} C_VEL
LIN {X 0,Y 530.999,Z 46.345,A -85,B 0,C 180,E1 -4474.942,E2 -4474.942} C_VEL
LIN {X 0,Y 530.976,Z 46.341,A -85,B 0,C 180,E1 -4478.247,E2 -4478.247} C_VEL
LIN {X 0,Y 530.99,Z 46.346,A -85,B 0,C 180,E1 -4480.677,E2 -4480.677} C_VEL
LIN {X 0,Y 530.986,Z 46.338,A -85,B 0,C 180,E1 -4483.071,E2 -4483.071} C_VEL
LIN {X 0,Y 531.024,Z 46.334,A -85,B 0,C 180,E1 -4485.436,E2 -4485.436} C_VEL
LIN {X 0,Y 531.042,Z 46.336,A -85,B 0,C 180,E1 -4488.55,E2 -4488.55} C_VEL
LIN {X 0,Y 531.057,Z 46.332,A -85,B 0,C 180,E1 -4491.629,E2 -4491.629} C_VEL
LIN {X 0,Y 531.123,Z 46.322,A -85,B 0,C 180,E1 -4494.685,E2 -4494.685} C_VEL
LIN {X 0,Y 531.142,Z 46.324,A -85,B 0,C 180,E1 -4497.725,E2 -4497.725} C_VEL
LIN {X 0,Y 531.156,Z 46.317,A -85,B 0,C 180,E1 -4500.758,E2 -4500.758} C_VEL
LIN {X 0,Y 531.106,Z 46.323,A -85,B 0,C 180,E1 -4503.034,E2 -4503.034} C_VEL
LIN {X 0,Y 531.055,Z 46.332,A -85,B 0,C 180,E1 -4506.077,E2 -4506.077} C_VEL
LIN {X 0,Y 531.019,Z 46.336,A -85,B 0,C 180,E1 -4509.138,E2 -4509.138} C_VEL
LIN {X 0,Y 531.045,Z 46.331,A -85,B 0,C 180,E1 -4512.225,E2 -4512.225} C_VEL
LIN {X 0,Y 531,Z 46.344,A -85,B 0,C 180,E1 -4515.35,E2 -4515.35} C_VEL
LIN {X 0,Y 530.981,Z 46.34,A -85,B 0,C 180,E1 -4518.521,E2 -4518.521} C_VEL
LIN {X 0,Y 531.003,Z 46.345,A -85,B 0,C 180,E1 -4520.938,E2 -4520.938} C_VEL
LIN {X 0,Y 530.973,Z 46.341,A -85,B 0,C 180,E1 -4524.225,E2 -4524.225} C_VEL
LIN {X 0,Y 530.991,Z 46.344,A -85,B 0,C 180,E1 -4526.744,E2 -4526.744} C_VEL
LIN {X 0,Y 530.983,Z 46.34,A -85,B 0,C 180,E1 -4529.322,E2 -4529.322} C_VEL
LIN {X 0,Y 530.968,Z 46.344,A -85,B 0,C 180,E1 -4532.1,E2 -4532.1} C_VEL
LIN {X 0,Y 530.967,Z 46.344,A -85,B 0,C 180,E1 -4534.85,E2 -4534.85} C_VEL
LIN {X 0,Y 530.966,Z 46.341,A -85,B 0,C 180,E1 -4537.508,E2 -4537.508} C_VEL
LIN {X 0,Y 530.967,Z 46.342,A -85,B 0,C 180,E1 -4540.434,E2 -4540.434} C_VEL
LIN {X 0,Y 530.946,Z 46.345,A -85,B 0,C 180,E1 -4543.279,E2 -4543.279} C_VEL
LIN {X 0,Y 530.945,Z 46.346,A -85,B 0,C 180,E1 -4543.553,E2 -4543.553} C_VEL
LIN {X 0,Y 530.272,Z 46.435,A -85,B 0,C 180,E1 -4544.186,E2 -4544.186} C_VEL
LIN {X 0,Y 527.417,Z 46.785,A -85,B 0,C 180,E1 -4545.215,E2 -4545.215} C_VEL
LIN {X 0,Y 525.008,Z 47.091,A -85,B 0,C 180,E1 -4546.044,E2 -4546.044} C_VEL
LIN {X 0,Y 523.975,Z 47.214,A -85,B 0,C 180,E1 -4546.683,E2 -4546.683} C_VEL
LIN {X 0,Y 523.893,Z 47.223,A -85,B 0,C 180,E1 -4546.9,E2 -4546.9} C_VEL
LIN {X 0,Y 523.938,Z 47.217,A -85,B 0,C 180,E1 -4548.907,E2 -4548.907} C_VEL
LIN {X 0,Y 523.913,Z 47.227,A -85,B 0,C 180,E1 -4551.898,E2 -4551.898} C_VEL
LIN {X 0,Y 523.923,Z 47.221,A -85,B 0,C 180,E1 -4554.911,E2 -4554.911} C_VEL
LIN {X 0,Y 523.936,Z 47.226,A -85,B 0,C 180,E1 -4557.68,E2 -4557.68} C_VEL
LIN {X 0,Y 523.953,Z 47.221,A -85,B 0,C 180,E1 -4560.677,E2 -4560.677} C_VEL
LIN {X 0,Y 523.999,Z 47.341,A -85,B 0,C 180,E1 -4561.621,E2 -4561.621} C_VEL
LIN {X 0,Y 524.481,Z 51.727,A -85,B 0,C 180,E1 -4562.548,E2 -4562.548} C_VEL
LIN {X 0,Y 524.302,Z 63.258,A -85,B 0,C 180,E1 -4564.905,E2 -4564.905} C_VEL
LIN {X 0,Y 526.024,Z 71.597,A -85,B 0,C 180,E1 -4565.08,E2 -4565.08} C_VEL
LIN {X 0,Y 525.561,Z 168.732,A -85,B 0,C 180,E1 -4566.427,E2 -4566.427} C_VEL
LIN {X 0,Y 525.418,Z 181.976,A -85,B 0,C 180,E1 -4566.759,E2 -4566.759} C_VEL
LIN {X 0,Y 525.282,Z 194.131,A -85,B 0,C 180,E1 -4567.217,E2 -4567.217} C_VEL
LIN {X 0,Y 524.973,Z 206.428,A -85,B 0,C 180,E1 -4567.841,E2 -4567.841} C_VEL
LIN {X 0,Y 524.677,Z 217.698,A -85,B 0,C 180,E1 -4568.592,E2 -4568.592} C_VEL
LIN {X 0,Y 524.447,Z 228.615,A -85,B 0,C 180,E1 -4569.507,E2 -4569.507} C_VEL
LIN {X 0,Y 524.166,Z 237.434,A -85,B 0,C 180,E1 -4570.415,E2 -4570.415} C_VEL
LIN {X 0,Y 523.955,Z 245.472,A -85,B 0,C 180,E1 -4571.424,E2 -4571.424} C_VEL
LIN {X 0,Y 523.794,Z 252.831,A -85,B 0,C 180,E1 -4572.56,E2 -4572.56} C_VEL
LIN {X 0,Y 523.642,Z 258.473,A -85,B 0,C 180,E1 -4573.629,E2 -4573.629} C_VEL
LIN {X 0,Y 523.513,Z 263.645,A -85,B 0,C 180,E1 -4574.864,E2 -4574.864} C_VEL
LIN {X 0,Y 523.459,Z 267.337,A -85,B 0,C 180,E1 -4576.015,E2 -4576.015} C_VEL
LIN {X 0,Y 523.384,Z 269.298,A -85,B 0,C 180,E1 -4576.804,E2 -4576.804} C_VEL
LIN {X 0,Y 523.382,Z 270.819,A -85,B 0,C 180,E1 -4577.593,E2 -4577.593} C_VEL
LIN {X 0,Y 523.364,Z 272.101,A -85,B 0,C 180,E1 -4578.603,E2 -4578.603} C_VEL
LIN {X 0,Y 523.342,Z 272.792,A -85,B 0,C 180,E1 -4579.946,E2 -4579.946} C_VEL
LIN {X 0,Y 523.323,Z 272.647,A -85,B 0,C 180,E1 -4580.726,E2 -4580.726} C_VEL
LIN {X 0,Y 523.371,Z 272.072,A -85,B 0,C 180,E1 -4581.506,E2 -4581.506} C_VEL
LIN {X 0,Y 523.459,Z 269.759,A -85,B 0,C 180,E1 -4583.06,E2 -4583.06} C_VEL
LIN {X 0,Y 523.498,Z 266.91,A -85,B 0,C 180,E1 -4584.221,E2 -4584.221} C_VEL
LIN {X 0,Y 523.558,Z 263.05,A -85,B 0,C 180,E1 -4585.38,E2 -4585.38} C_VEL
LIN {X 0,Y 523.653,Z 258.08,A -85,B 0,C 180,E1 -4586.538,E2 -4586.538} C_VEL
LIN {X 0,Y 523.744,Z 251.857,A -85,B 0,C 180,E1 -4587.693,E2 -4587.693} C_VEL
LIN {X 0,Y 523.989,Z 244.068,A -85,B 0,C 180,E1 -4588.847,E2 -4588.847} C_VEL
LIN {X 0,Y 524.217,Z 234.419,A -85,B 0,C 180,E1 -4590,E2 -4590} C_VEL
LIN {X 0,Y 524.502,Z 224.378,A -85,B 0,C 180,E1 -4590.96,E2 -4590.96} C_VEL
LIN {X 0,Y 524.819,Z 213.055,A -85,B 0,C 180,E1 -4591.823,E2 -4591.823} C_VEL
LIN {X 0,Y 525.123,Z 201.932,A -85,B 0,C 180,E1 -4592.493,E2 -4592.493} C_VEL
LIN {X 0,Y 525.311,Z 190.663,A -85,B 0,C 180,E1 -4593.02,E2 -4593.02} C_VEL
LIN {X 0,Y 525.469,Z 177.809,A -85,B 0,C 180,E1 -4593.451,E2 -4593.451} C_VEL
LIN {X 0,Y 525.601,Z 164.075,A -85,B 0,C 180,E1 -4593.738,E2 -4593.738} C_VEL
LIN {X 0,Y 525.879,Z 71.126,A -85,B 0,C 180,E1 -4595.02,E2 -4595.02} C_VEL
LIN {X 0,Y 524.273,Z 63.127,A -85,B 0,C 180,E1 -4595.192,E2 -4595.192} C_VEL
LIN {X 0,Y 524.54,Z 51.87,A -85,B 0,C 180,E1 -4597.483,E2 -4597.483} C_VEL
LIN {X 0,Y 524.002,Z 47.217,A -85,B 0,C 180,E1 -4598.484,E2 -4598.484} C_VEL
LIN {X 0,Y 524.005,Z 47.207,A -85,B 0,C 180,E1 -4601.74,E2 -4601.74} C_VEL
LIN {X 0,Y 523.996,Z 47.211,A -85,B 0,C 180,E1 -4605.053,E2 -4605.053} C_VEL
LIN {X 0,Y 523.966,Z 47.215,A -85,B 0,C 180,E1 -4607.969,E2 -4607.969} C_VEL
LIN {X 0,Y 523.974,Z 47.22,A -85,B 0,C 180,E1 -4610.41,E2 -4610.41} C_VEL
LIN {X 0,Y 523.913,Z 47.221,A -85,B 0,C 180,E1 -4612.894,E2 -4612.894} C_VEL
LIN {X 0,Y 523.987,Z 47.217,A -85,B 0,C 180,E1 -4616.02,E2 -4616.02} C_VEL
LIN {X 0,Y 523.942,Z 47.216,A -85,B 0,C 180,E1 -4618.875,E2 -4618.875} C_VEL
LIN {X 0,Y 523.923,Z 47.221,A -85,B 0,C 180,E1 -4621.544,E2 -4621.544} C_VEL
LIN {X 0,Y 523.944,Z 47.218,A -85,B 0,C 180,E1 -4624.29,E2 -4624.29} C_VEL
LIN {X 0,Y 523.913,Z 47.22,A -85,B 0,C 180,E1 -4627.132,E2 -4627.132} C_VEL
LIN {X 0,Y 523.94,Z 47.218,A -85,B 0,C 180,E1 -4630.13,E2 -4630.13} C_VEL
LIN {X 0,Y 523.938,Z 47.216,A -85,B 0,C 180,E1 -4632.459,E2 -4632.459} C_VEL
LIN {X 0,Y 523.945,Z 47.222,A -85,B 0,C 180,E1 -4635.311,E2 -4635.311} C_VEL
LIN {X 0,Y 523.959,Z 47.215,A -85,B 0,C 180,E1 -4638.69,E2 -4638.69} C_VEL
LIN {X 0,Y 523.921,Z 47.225,A -85,B 0,C 180,E1 -4641.081,E2 -4641.081} C_VEL
LIN {X 0,Y 523.904,Z 47.221,A -85,B 0,C 180,E1 -4643.826,E2 -4643.826} C_VEL
LIN {X 0,Y 523.946,Z 47.218,A -85,B 0,C 180,E1 -4646.636,E2 -4646.636} C_VEL
LIN {X 0,Y 523.96,Z 47.217,A -85,B 0,C 180,E1 -4649.356,E2 -4649.356} C_VEL
LIN {X 0,Y 523.982,Z 47.212,A -85,B 0,C 180,E1 -4652.282,E2 -4652.282} C_VEL
LIN {X 0,Y 523.952,Z 47.22,A -85,B 0,C 180,E1 -4654.581,E2 -4654.581} C_VEL
LIN {X 0,Y 523.924,Z 47.218,A -85,B 0,C 180,E1 -4657.757,E2 -4657.757} C_VEL
LIN {X 0,Y 523.975,Z 47.218,A -85,B 0,C 180,E1 -4660.408,E2 -4660.408} C_VEL
LIN {X 0,Y 523.951,Z 47.218,A -85,B 0,C 180,E1 -4662.837,E2 -4662.837} C_VEL
LIN {X 0,Y 523.983,Z 47.211,A -85,B 0,C 180,E1 -4665.236,E2 -4665.236} C_VEL
LIN {X 0,Y 524.019,Z 47.213,A -85,B 0,C 180,E1 -4668.394,E2 -4668.394} C_VEL
LIN {X 0,Y 523.993,Z 47.21,A -85,B 0,C 180,E1 -4671.516,E2 -4671.516} C_VEL
LIN {X 0,Y 524.05,Z 47.208,A -85,B 0,C 180,E1 -4673.841,E2 -4673.841} C_VEL
LIN {X 0,Y 524.047,Z 47.202,A -85,B 0,C 180,E1 -4676.925,E2 -4676.925} C_VEL
LIN {X 0,Y 524.119,Z 47.2,A -85,B 0,C 180,E1 -4680,E2 -4680} C_VEL
LIN {X 0,Y 524.074,Z 47.2,A -85,B 0,C 180,E1 -4683.075,E2 -4683.075} C_VEL
LIN {X 0,Y 524.016,Z 47.208,A -85,B 0,C 180,E1 -4686.159,E2 -4686.159} C_VEL
LIN {X 0,Y 523.994,Z 47.209,A -85,B 0,C 180,E1 -4688.484,E2 -4688.484} C_VEL
LIN {X 0,Y 524.006,Z 47.212,A -85,B 0,C 180,E1 -4691.738,E2 -4691.738} C_VEL
LIN {X 0,Y 523.999,Z 47.214,A -85,B 0,C 180,E1 -4695.052,E2 -4695.052} C_VEL
LIN {X 0,Y 523.951,Z 47.215,A -85,B 0,C 180,E1 -4697.97,E2 -4697.97} C_VEL
LIN {X 0,Y 523.978,Z 47.212,A -85,B 0,C 180,E1 -4700.41,E2 -4700.41} C_VEL
LIN {X 0,Y 523.916,Z 47.226,A -85,B 0,C 180,E1 -4702.893,E2 -4702.893} C_VEL
LIN {X 0,Y 523.935,Z 47.219,A -85,B 0,C 180,E1 -4705.42,E2 -4705.42} C_VEL
LIN {X 0,Y 523.93,Z 47.217,A -85,B 0,C 180,E1 -4708.001,E2 -4708.001} C_VEL
LIN {X 0,Y 523.95,Z 47.222,A -85,B 0,C 180,E1 -4710.855,E2 -4710.855} C_VEL
LIN {X 0,Y 523.934,Z 47.217,A -85,B 0,C 180,E1 -4713.729,E2 -4713.729} C_VEL
LIN {X 0,Y 523.903,Z 47.227,A -85,B 0,C 180,E1 -4716.401,E2 -4716.401} C_VEL
LIN {X 0,Y 523.923,Z 47.219,A -85,B 0,C 180,E1 -4719.085,E2 -4719.085} C_VEL
LIN {X 0,Y 523.956,Z 47.22,A -85,B 0,C 180,E1 -4722.119,E2 -4722.119} C_VEL
LIN {X 0,Y 523.942,Z 47.216,A -85,B 0,C 180,E1 -4725.311,E2 -4725.311} C_VEL
LIN {X 0,Y 523.957,Z 47.215,A -85,B 0,C 180,E1 -4728.69,E2 -4728.69} C_VEL
LIN {X 0,Y 523.917,Z 47.226,A -85,B 0,C 180,E1 -4731.898,E2 -4731.898} C_VEL
LIN {X 0,Y 523.926,Z 47.218,A -85,B 0,C 180,E1 -4734.911,E2 -4734.911} C_VEL
LIN {X 0,Y 523.938,Z 47.224,A -85,B 0,C 180,E1 -4737.68,E2 -4737.68} C_VEL
LIN {X 0,Y 523.957,Z 47.216,A -85,B 0,C 180,E1 -4740.677,E2 -4740.677} C_VEL
LIN {X 0,Y 523.975,Z 47.218,A -85,B 0,C 180,E1 -4743.728,E2 -4743.728} C_VEL
LIN {X 0,Y 523.998,Z 47.304,A -85,B 0,C 180,E1 -4744.716,E2 -4744.716} C_VEL
LIN {X 0,Y 525.401,Z 54.937,A -85,B 0,C 180,E1 -4745.922,E2 -4745.922} C_VEL
LIN {X 0,Y 525.094,Z 70.299,A -85,B 0,C 180,E1 -4748.197,E2 -4748.197} C_VEL
LIN {X 0,Y 524.751,Z 89.761,A -85,B 0,C 180,E1 -4751.047,E2 -4751.047} C_VEL
LIN {X 0,Y 524.341,Z 109.146,A -85,B 0,C 180,E1 -4753.852,E2 -4753.852} C_VEL
LIN {X 0,Y 524.184,Z 115.878,A -85,B 0,C 180,E1 -4754.819,E2 -4754.819} C_VEL
LIN {X 0,Y 525.897,Z 127.989,A -85,B 0,C 180,E1 -4755.05,E2 -4755.05} C_VEL
LIN {X 0,Y 525.476,Z 224.621,A -85,B 0,C 180,E1 -4756.39,E2 -4756.39} C_VEL
LIN {X 0,Y 525.216,Z 237.967,A -85,B 0,C 180,E1 -4756.728,E2 -4756.728} C_VEL
LIN {X 0,Y 524.982,Z 250.185,A -85,B 0,C 180,E1 -4757.19,E2 -4757.19} C_VEL
LIN {X 0,Y 524.731,Z 261.53,A -85,B 0,C 180,E1 -4757.763,E2 -4757.763} C_VEL
LIN {X 0,Y 524.458,Z 272.863,A -85,B 0,C 180,E1 -4758.502,E2 -4758.502} C_VEL
LIN {X 0,Y 524.204,Z 283.576,A -85,B 0,C 180,E1 -4759.377,E2 -4759.377} C_VEL
LIN {X 0,Y 523.903,Z 293.229,A -85,B 0,C 180,E1 -4760.347,E2 -4760.347} C_VEL
LIN {X 0,Y 523.707,Z 301.148,A -85,B 0,C 180,E1 -4761.317,E2 -4761.317} C_VEL
LIN {X 0,Y 523.558,Z 308.887,A -85,B 0,C 180,E1 -4762.479,E2 -4762.479} C_VEL
LIN {X 0,Y 523.431,Z 316.021,A -85,B 0,C 180,E1 -4763.834,E2 -4763.834} C_VEL
LIN {X 0,Y 523.382,Z 320.769,A -85,B 0,C 180,E1 -4764.993,E2 -4764.993} C_VEL
LIN {X 0,Y 523.443,Z 324.402,A -85,B 0,C 180,E1 -4766.151,E2 -4766.151} C_VEL
LIN {X 0,Y 523.417,Z 326.272,A -85,B 0,C 180,E1 -4766.921,E2 -4766.921} C_VEL
LIN {X 0,Y 523.338,Z 327.671,A -85,B 0,C 180,E1 -4767.691,E2 -4767.691} C_VEL
LIN {X 0,Y 523.279,Z 329.279,A -85,B 0,C 180,E1 -4769.23,E2 -4769.23} C_VEL
LIN {X 0,Y 523.283,Z 329.495,A -85,B 0,C 180,E1 -4770,E2 -4770} C_VEL
LIN {X 0,Y 523.279,Z 329.276,A -85,B 0,C 180,E1 -4770.769,E2 -4770.769} C_VEL
LIN {X 0,Y 523.338,Z 327.664,A -85,B 0,C 180,E1 -4772.309,E2 -4772.309} C_VEL
LIN {X 0,Y 523.417,Z 326.262,A -85,B 0,C 180,E1 -4773.079,E2 -4773.079} C_VEL
LIN {X 0,Y 523.422,Z 323.306,A -85,B 0,C 180,E1 -4774.235,E2 -4774.235} C_VEL
LIN {X 0,Y 523.453,Z 319.307,A -85,B 0,C 180,E1 -4775.393,E2 -4775.393} C_VEL
LIN {X 0,Y 523.486,Z 313.254,A -85,B 0,C 180,E1 -4776.728,E2 -4776.728} C_VEL
LIN {X 0,Y 523.635,Z 306.441,A -85,B 0,C 180,E1 -4777.907,E2 -4777.907} C_VEL
LIN {X 0,Y 523.774,Z 298.11,A -85,B 0,C 180,E1 -4779.071,E2 -4779.071} C_VEL
LIN {X 0,Y 523.977,Z 289.576,A -85,B 0,C 180,E1 -4780.042,E2 -4780.042} C_VEL
LIN {X 0,Y 524.285,Z 279.039,A -85,B 0,C 180,E1 -4781.012,E2 -4781.012} C_VEL
LIN {X 0,Y 524.55,Z 267.427,A -85,B 0,C 180,E1 -4781.871,E2 -4781.871} C_VEL
LIN {X 0,Y 524.859,Z 255.264,A -85,B 0,C 180,E1 -4782.568,E2 -4782.568} C_VEL
LIN {X 0,Y 525.131,Z 242.872,A -85,B 0,C 180,E1 -4783.102,E2 -4783.102} C_VEL
LIN {X 0,Y 525.379,Z 230.153,A -85,B 0,C 180,E1 -4783.489,E2 -4783.489} C_VEL
LIN {X 0,Y 525.551,Z 215.035,A -85,B 0,C 180,E1 -4783.756,E2 -4783.756} C_VEL
LIN {X 0,Y 525.81,Z 127.366,A -85,B 0,C 180,E1 -4784.96,E2 -4784.96} C_VEL
LIN {X 0,Y 524.225,Z 115.744,A -85,B 0,C 180,E1 -4785.187,E2 -4785.187} C_VEL
LIN {X 0,Y 524.674,Z 94.098,A -85,B 0,C 180,E1 -4788.307,E2 -4788.307} C_VEL
LIN {X 0,Y 525.03,Z 74.421,A -85,B 0,C 180,E1 -4791.187,E2 -4791.187} C_VEL
LIN {X 0,Y 525.458,Z 55.053,A -85,B 0,C 180,E1 -4794.075,E2 -4794.075} C_VEL
LIN {X 0,Y 523.996,Z 47.215,A -85,B 0,C 180,E1 -4795.363,E2 -4795.363} C_VEL
LIN {X 0,Y 523.968,Z 47.22,A -85,B 0,C 180,E1 -4797.999,E2 -4797.999} C_VEL
LIN {X 0,Y 523.948,Z 47.217,A -85,B 0,C 180,E1 -4800.855,E2 -4800.855} C_VEL
LIN {X 0,Y 523.934,Z 47.222,A -85,B 0,C 180,E1 -4803.73,E2 -4803.73} C_VEL
LIN {X 0,Y 523.907,Z 47.224,A -85,B 0,C 180,E1 -4806.401,E2 -4806.401} C_VEL
LIN {X 0,Y 523.923,Z 47.217,A -85,B 0,C 180,E1 -4809.085,E2 -4809.085} C_VEL
LIN {X 0,Y 523.955,Z 47.218,A -85,B 0,C 180,E1 -4812.119,E2 -4812.119} C_VEL
LIN {X 0,Y 523.946,Z 47.218,A -85,B 0,C 180,E1 -4815.31,E2 -4815.31} C_VEL
LIN {X 0,Y 523.959,Z 47.213,A -85,B 0,C 180,E1 -4818.69,E2 -4818.69} C_VEL
LIN {X 0,Y 523.921,Z 47.22,A -85,B 0,C 180,E1 -4821.081,E2 -4821.081} C_VEL
LIN {X 0,Y 523.904,Z 47.222,A -85,B 0,C 180,E1 -4823.825,E2 -4823.825} C_VEL
LIN {X 0,Y 523.917,Z 47.219,A -85,B 0,C 180,E1 -4826.634,E2 -4826.634} C_VEL
LIN {X 0,Y 523.96,Z 47.217,A -85,B 0,C 180,E1 -4829.356,E2 -4829.356} C_VEL
LIN {X 0,Y 523.981,Z 47.212,A -85,B 0,C 180,E1 -4832.281,E2 -4832.281} C_VEL
LIN {X 0,Y 523.951,Z 47.218,A -85,B 0,C 180,E1 -4834.581,E2 -4834.581} C_VEL
LIN {X 0,Y 523.924,Z 47.217,A -85,B 0,C 180,E1 -4837.757,E2 -4837.757} C_VEL
LIN {X 0,Y 523.974,Z 47.217,A -85,B 0,C 180,E1 -4840.408,E2 -4840.408} C_VEL
LIN {X 0,Y 523.969,Z 47.215,A -85,B 0,C 180,E1 -4842.837,E2 -4842.837} C_VEL
LIN {X 0,Y 523.982,Z 47.211,A -85,B 0,C 180,E1 -4845.236,E2 -4845.236} C_VEL
LIN {X 0,Y 524.018,Z 47.212,A -85,B 0,C 180,E1 -4848.394,E2 -4848.394} C_VEL
LIN {X 0,Y 524.005,Z 47.209,A -85,B 0,C 180,E1 -4851.516,E2 -4851.516} C_VEL
